// TwinCAT 3 PLC project PulsePower_PLC
// ProgramVersion: 3.1.4023.0
// libraries:
//   Tc2_BACnetRev12, * (Beckhoff Automation GmbH)
//   Tc2_DataExchange, * (Beckhoff Automation GmbH)
//   Tc2_Math, * (Beckhoff Automation GmbH)
//   Tc2_NC, * (Beckhoff Automation GmbH)
//   Tc2_Standard, * (Beckhoff Automation GmbH)
//   Tc2_System, * (Beckhoff Automation GmbH)
//   Tc3_EventLogger, * (Beckhoff Automation GmbH)
//   Tc3_Module, * (Beckhoff Automation GmbH)
// project tree:
//   DUTs/ E_Command.TcDUT (not stored), E_PulseState.TcDUT (not stored), E_Status.TcDUT (not stored), ST_Alarm_Base.TcDUT, ST_Charger_Base.TcDUT (not stored), ST_ChargeTime.TcDUT, ST_Control.TcDUT (not stored), ST_Echo_MCP.TcDUT, ST_Echo_Section.TcDUT (not stored), ST_FieldDevices_Base.TcDUT (not stored), ST_FieldDevices_Form.TcDUT, ST_InstrumentReading.TcDUT (not stored), ST_Recipe.TcDUT (not stored), ST_RelayFaults_Base.TcDUT, ST_RelayFaults_Form.TcDUT, ST_Section_Base.TcDUT, ST_Setpoints_Base.TcDUT, ST_Trip_Base.TcDUT, ST_VoltageFeedback.TcDUT
//   GVLs/ Alarms_DB.TcGVL (not stored), ChargeTime_DB.TcGVL, Command.TcGVL, EngVal.TcGVL, GVL.TcGVL, Recipe.TcGVL, Setpoints.TcGVL (not stored), TxMainPLC.TcGVL, HMI_DB.TcGVL, Input.TcGVL (not stored), InstrumentReading.TcGVL (not stored), LCP.TcGVL, MCP_IO.TcGVL (not stored), Output.TcGVL (not stored), Permissives_DB.TcGVL (not stored), Trips_DB.TcGVL (not stored)
//   / PlcTask.TcTTO (not stored)
//   POUs/ ADC_10V.TcPOU (not stored), ADC_5V.TcPOU (not stored), Alarms.TcPOU, Alarms_FB.TcPOU (not stored), Alias.TcPOU (not stored), AnalogConversion.TcPOU, AQ.TcPOU (not stored), ChargeTime.TcPOU, Communication.TcPOU (not stored), Dump_FB.TcPOU, Heartbeat.TcPOU (not stored), HMI.TcPOU, LCA_CAL.TcPOU (not stored), MAIN.TcPOU, Norm_x.TcPOU (not stored), Permissives.TcPOU, PWMO.TcPOU (not stored), Sequence.TcPOU, Trips.TcPOU
// real-time tasks:
//   TASK PlcTask: cycle T#10ms, priority 20, ADS port 350
// I/O:
//   DEVICE Device 3 (EtherCAT) (disabled), AmsNetId 5.104.224.86.4.1
//   DEVICE Device 1 (EL6751) (disabled), AmsNetId 5.104.224.86.2.1
//   DEVICE Device 2 (EtherCAT), AmsNetId 5.104.224.86.3.1
//     Term 1 (EK1200) [EK1200-5000 EtherCAT Power supply (2A E-Bus)]
//       Term 9 (EL2008) [EL2008 8Ch. Dig. Output 24V, 0.5A]
//       Term 3 (EL9011) [EL9011 End Terminal]
// variable links:
//   PulsePower_PLC/PulsePower_PLC Instance <-> Device 2 (EtherCAT)/Term 1 (EK1200)/Term 9 (EL2008)
//     PlcTask Outputs/Output.R2_01_00 <-> Channel 1/Output

// ---- DUTs/ST_Alarm_Base.TcDUT
TYPE ST_Alarm_Base :
STRUCT
	AlarmWord : WORD;
END_STRUCT
END_TYPE

// ---- DUTs/ST_ChargeTime.TcDUT
TYPE ST_ChargeTime :
STRUCT
	timeToChargeLoad : REAL;
	Power			 : REAL;
END_STRUCT
END_TYPE

// ---- DUTs/ST_Echo_MCP.TcDUT
TYPE ST_Echo_MCP :
STRUCT
	VoltageFeedback : REAL; //DINT;
	CurrentFeedback : REAL; //DINT;
	TDKLoad			: ST_ChargeTime;
	
END_STRUCT
END_TYPE

// ---- DUTs/ST_FieldDevices_Form.TcDUT
TYPE ST_FieldDevices_Form EXTENDS ST_FieldDevices_Base :
STRUCT
	PreFormChargeRly_close		: BOOL;
	FormTrigChargeRly_close		: BOOL;
	PreFormTrigChargeRly_close 	: BOOL;
	PreFormDumpRly_close		: BOOL;
	FormTrigDumpRly1_close		: BOOL;
	PreFormTrigDumpRly1_close	: BOOL;
	
	ClosePreFormChargeRly		: BOOL;
	CloseFormTrigChargeRly		: BOOL;
	ClosePreFormTrigChargeRly	: BOOL;
	OpenPreFormDumpRly			: BOOL;
	OpenFormTrigDumpRly1		: BOOL;
	OpenPreFormTrigDumpRly1		: BOOL;
	
	FormTrigShortContact_close		: BOOL;
	FormTrigUnshortContact_close	: BOOL;
	FormTrigShortContactEngaged		: BOOL;
	FormTrigShortContactUnknown		: BOOL;
	
	PreFormTrigShortContact_close 	: BOOL;
	PreFormTrigUnShortContact_close : BOOL;
	PreFormTrigShortContactEngaged	: BOOL;
	PreFormTrigShortContactUnknown	: BOOL;
	

END_STRUCT
END_TYPE

// ---- DUTs/ST_RelayFaults_Base.TcDUT
TYPE ST_RelayFaults_Base :
STRUCT
	DumpRelay1_FailtoClose		: BOOL;
	DumpRelay1_FailtoOpen		: BOOL;
	DumpRelay1_Failed			: BOOL;
	DumpRly1FaultDelay_TON 		: TON;
	DumpRly2FaultDelay_TON 		: TON;
	
	DumpRelay2_FailtoClose		: BOOL;
	DumpRelay2_FailtoOpen		: BOOL;
	DumpRelay2_Failed			: BOOL;
	
	ChargeRelay1_FailtoClose	: BOOL;
	ChargeRelay1_FailtoOpen		: BOOL;
	ChargeRelay1_Failed			: BOOL;
	ChrgRly1FaultDelay_TON	 	: TON;
	
	ChargeRelay2_FailtoClose	: BOOL;
	ChargeRelay2_FailtoOpen		: BOOL;
	ChargeRelay2_Failed			: BOOL;
	ChrgRly2FaultDelay_TON	 	: TON;
	

END_STRUCT
END_TYPE

// ---- DUTs/ST_RelayFaults_Form.TcDUT
TYPE ST_RelayFaults_Form EXTENDS ST_RelayFaults_Base :
STRUCT
	PreFormChrgRlyFailed				: BOOL;
	PreFormChrgRlyFaultDelay_TON		: TON;
	FormTrigChrgRlyFailed				: BOOL;
	FormTrigChrgRlyFaultDelay_TON		: TON;
	PreFormTrigChrgRlyFailed			: BOOL;
	PreFormTrigChrgRlyFaultDelay_TON	: TON;
	PreFormDumpRlyFailed				: BOOL;
	PreFormDumpRlyFaultDelay_TON		: TON;
	FormTrigDumpRly1Failed				: BOOL;
	FormTrigDumpRlyFaultDelay_TON		: TON;
	PreFormTrigDumpRly1Failed			: BOOL;
	PreFormTrigDumpRlyFaultDelay_TON	: TON;
	
END_STRUCT
END_TYPE

// ---- DUTs/ST_Section_Base.TcDUT
//Base coil type with all the Common functionality
TYPE ST_Section_Base :
STRUCT
	
	Peak : ST_FieldDevices_Base;
	Sust : ST_FieldDevices_Base;
	Form : ST_FieldDevices_Form;
	
	PreFormCapVoltage_raw			: INT;
	PreFormCapVoltage_norm			: REAL;
	PreFormCapVoltageFeedback		: REAL;
	
	FormTriggerVoltage_raw			: INT;
	FormTriggerVoltage_norm			: REAL;
	FormTriggerVoltageFeedback		: REAL;
	
	PreFormTriggerVoltage_raw		: INT;
	PreFormTriggerVoltage_norm		: REAL;
	PreFormTriggerVoltageFeedback	: REAL;
	
	PreFormCapDischarged			: BOOL;
	PreFormCapFullyChaged			: BOOL;
	
	PSU1_DCOK						: BOOL := FALSE;
	//Local_EstopPB_Pressed			: BOOL;  //NC
	SystemReadyToCharge				: BOOL := FALSE;
	LossPneumaticPressure			: BOOL;
	AllCapsDischarged				: BOOL;
	AllCapsFullyCharged				: BOOL;
	//PreFormBank						: ST_ChargeTime;
END_STRUCT
END_TYPE

// ---- DUTs/ST_Setpoints_Base.TcDUT
TYPE ST_Setpoints_Base :
STRUCT
	RequiredChargedV : REAL := 12;
	TotalCapacitance : REAL := 10; //uF - LOCAL ONLY, NOT FROM MAIN PLC - LoadCapacitance
	PSratedV		 : REAL := 50;
	wLCA			 : BOOL := TRUE;
	NumOfCharger	 : INT := 1;
END_STRUCT
END_TYPE

// ---- DUTs/ST_Trip_Base.TcDUT
TYPE ST_Trip_Base :
STRUCT
	ChargerVoltageReadingFaulted 		: BOOL;
	CurrentReadingFaulted 		 		: BOOL;
	
	//ACInterlockRelayFailedtoClose		: BOOL;
	//ACInterlockRelayFailedtoOpen 		: BOOL;
	//ACintLockRlyCloseFaultDelay_TON	: TON;
	//ACintLockRlyOpenFaultDelay_TON	: TON;
	
	Peak 								: ST_RelayFaults_Base;
	Sust 								: ST_RelayFaults_Base;
	Form 								: ST_RelayFaults_Form;
	
	SystemTripped						: BOOL;
	LossPneumaticPressure				: BOOL;
	LossDCPower							: BOOL;
	
	(*HVisoRelayFailedToOpen		: BOOL;
	HVRelayOpenFaultDelay_TON	: TON;
	HVisoRelayFailedToClose		: BOOL;
	HVRelayCloseFaultDelay_TON	: TON;
	*)
END_STRUCT
END_TYPE

// ---- DUTs/ST_VoltageFeedback.TcDUT
TYPE ST_VoltageFeedback :
STRUCT
	voltageFeedback_raw : INT;
END_STRUCT
END_TYPE

// ---- GVLs/ChargeTime_DB.TcGVL
{attribute 'qualified_only'}
VAR_GLOBAL RETAIN
	ChargerDelay_TON : ARRAY[1..8] OF TON;
	ChargerDelay_PT  : ARRAY[1..8] OF TIME;
	ChargerDelay_ET  : ARRAY[1..8] OF TIME;	
	
	//SustChargeTime_TON : ARRAY[1..3] OF TON;
	//SustChargeTime_PT  : ARRAY[1..3] OF TIME;
	//SustChargeTime_ET  : ARRAY[1..3] OF TIME;	
	
	//FormChargeTime_TON : ARRAY[1..2] OF TON;
	//FormChargeTime_PT  : ARRAY[1..2] OF TIME;
	//FormChargeTime_ET  : ARRAY[1..2] OF TIME;
	
	PreFormChargeTime_TON : TON;
	PreFormChargeTime_PT : TIME;
	PreFormChargeTime_ET : TIME;
	
	LongestChargeTime_TON : TON;
	LongestChargeTime_PT : TIME;
	LongestChargeTime_ET : TIME;

	ChargeTimeStartDelay	: ARRAY[1..8] OF INT;
	ChargingTimeElapse		: ARRAY[1..8] OF INT;	
	ChargingTimeElapse_TON	: ARRAY[1..8] OF TON;
	
	PreFormChargeTimeStartDelay : INT;
	PreFormChargingTimeElapse : INT;
	PreFormChargingTimeElapse_TON : TON;
END_VAR

// ---- GVLs/Command.TcGVL
{attribute 'qualified_only'}
VAR_GLOBAL
	eCommand : E_Command;
END_VAR

// ---- GVLs/EngVal.TcGVL
{attribute 'qualified_only'}
VAR_GLOBAL
	Max_50kVChargerVoltage : REAL := 50000; //50kV
	Min_50kVChargerVoltage : REAL := 0;
	
	Max_50kVChargerCurrent : REAL := 0.18; //total peak charge current is 0.18A
	Min_50kVChargerCurrent : REAL := 0;
	
	Max_12kVChargerVoltage : REAL := 12000; //12kV
	Min_12kVChargerVoltage : REAL := 0;
	
	Max_12kVChargerCurrent : REAL := 0.75; //total peak charge current is 0.75A
	Min_12kVChargerCurrent : REAL := 0;
	
	Max_GLS1_ChargerV	   : REAL := 50000; //form trigger
	Max_GLS2_ChargerV	   : REAL := 50000; // preform trigger
	Max_GLS3_ChargerV	   : REAL := 30000; // preform cap charger
	
	Max_CapVoltage			: REAL := 32000;  //assuming 32kV cap....  
	Min_CapVoltage			: REAL := 0;
	
	UpperLimit12kVCaps		: REAL := 10000; //peak and sust
	//LowerLimit12kVCaps	: REAL := -2000;
	UpperLimit50kVCaps		: REAL := 35000; //formation
	
	(*ULimit_PeakCapRequiredV	: REAL := 10000; //10kV veto
	LLimit_PeakCapRequiredV	: REAL := -2000; //-2kV
	ULimit_SustCapRequiredV	: REAL := 12000; //12kv veto
	LLimit_SustCapRequiredV	: REAL := -2000; //-2kv
	ULimit_FormCapRequiredV : REAL := 35000;
	LLimit_FormCapRequiredV : REAL := 0;
	*)
	ULimit_PreFormCapRequiredV : REAL := 30000; //gls3
	LLimit_PreFormCapRequiredV : REAL := 0;
		
END_VAR

// ---- GVLs/GVL.TcGVL
{attribute 'qualified_only'}
VAR_GLOBAL
	alarm_test	: BOOL;
	test		: BOOL;
	RemoteModeSelected : BOOL;
END_VAR

// ---- GVLs/Recipe.TcGVL
{attribute 'qualified_only'}
VAR_GLOBAL
	TDKLoad : ARRAY [1..8] OF ST_Recipe;
	GLSLoad : ST_Recipe;
	GLS1_VSP : REAL := 50; //DINT;
	GLS2_VSP : REAL := 50; //DINT;
	PeakSupplyEN	: BOOL := TRUE;
	SustSupplyEN	: BOOL := TRUE;
	FormSupplyEN	: BOOL := TRUE;
	PFormSupplyEN	: BOOL := TRUE;
END_VAR

// ---- GVLs/TxMainPLC.TcGVL
{attribute 'qualified_only'}
VAR_GLOBAL
	Charger		: ARRAY[1..8] OF ST_Echo_MCP;
	GLSLoad		: ST_ChargeTime;
	Section 	: ARRAY[1..4] OF ST_Echo_Section;
	ChargeRunOutTime	: REAL; //DINT;
	ChargingRunOutTime	: REAL; //DINT;
END_VAR

// ---- GVLs/HMI_DB.TcGVL
{attribute 'qualified_only'}
VAR_GLOBAL PERSISTENT
	RemoteModeSelected 	: BOOL := TRUE;
	
	OpenAllDumpRlyPB	: BOOL;
	CloseAllChargeRlyPB	: BOOL;
	AbortPB				: BOOL;
	
	ChargerHVOFF_rlyDelayPT		: TIME := T#25MS;
	ChargerHVOFF_rlyDelayPT_INT	: INT := 25;
	
	HVONdelayPT					: TIME := T#250MS;
	HVONdelayPT_INT				: INT := 250;
	
	RunOutTMR_PT				: TIME := T#10S;
	RunOutTMR_PT_INT			: INT := 10;
	RunOutTMR_elapse			: INT;
	
	ChargingRunOutTMR_elapse	: INT;
	
	//admin bypasses
	SafetyOKBP					: BOOL;
	AllDumpRelaysOpenBP			: BOOL;
	InterlockPressureLossBP		: BOOL;
	AllChargeRelayCloseBP		: BOOL;
	NoFaultDetectedBP			: BOOL;
	//AllShortingSysRemovedBP		: BOOL;
	AlldcPSUokBP				: BOOL;
	LossHVsignalBP				: BOOL;
	
	//timeToChargeLoad 			: ARRAY [1..8] OF REAL;
	//GLSchargeTime	 			: ARRAY [1..3] OF REAL;
	TDKLoad 					: ARRAY [1..8] OF ST_Setpoints_Base; //or RETAIN
	GLSLoad	 					: ST_Setpoints_Base;
	
	(*PSratedV					: REAL := 50;
	RequiredChargeV				: REAL := 30;
	LoadCapacitance				: REAL := 600;
	wLCA						: BOOL := TRUE;
	NumOfCharger				: INT := 1;*)
END_VAR

VAR_GLOBAL
	LiftMachineGNDsw			: BOOL := FALSE;
	//for startup run
	PeakChargerSP				: DINT;
	SustChargerSP				: DINT;
	FormChargerSP				: DINT;
	PreFormChargerSP			: DINT;
	FormTrigChargerSP			: DINT;
	PreFormTrigChargerSP		: DINT;
	
	OpenAllPeakDumpRlySW		: BOOL := FALSE;
	OpenAllSustDumpRlySW		: BOOL := FALSE;
	OpenAllFormDumpRlySW		: BOOL := FALSE;
	OpenAllPreFormDumpRlySW		: BOOL := FALSE;
	OpenFormTrigDumpRlySW		: BOOL := FALSE;
	OpenPreFormTrigDumpRlySW	: BOOL := FALSE;
	
	CloseAllPeakChargRlySW		: BOOL := FALSE;
	CloseAllSustChargRlySW		: BOOL := FALSE;
	CloseAllFormChargRlySW		: BOOL := FALSE;
	CloseAllPreFormChargRlySW	: BOOL := FALSE;
	CloseFormTrigChargeRlySW	: BOOL := FALSE;
	ClosePreFormTrigChargeRlySW : BOOL := FALSE;
	
	PeakHVONsw					: BOOL := FALSE; //enable
	SustHVONsw					: BOOL := FALSE; //enable
	FormHVONsw					: BOOL := FALSE; //enable
	PreFormHVONsw				: BOOL := FALSE;
	GLS1HVONsw					: BOOL := FALSE;
	GLS2HVONsw					: BOOL := FALSE;
	
	DumpALLPB_Local				: BOOL := FALSE;
	
	(*PeakInhibitONsw				: BOOL;
	SustInhibitONsw				: BOOL;
	FormInhibitONsw				: BOOL;
	PreFormInhibitONsw			: BOOL;
	*)	
END_VAR

// ---- GVLs/LCP.TcGVL
{attribute 'qualified_only'}
VAR_GLOBAL
	Section : ARRAY [1..4] OF ST_Section_Base;
END_VAR

// ---- POUs/Alarms.TcPOU
PROGRAM Alarms
VAR
	bWarning : BOOL;
	bConfirm : BOOL;
	alarms : ARRAY[0..128] OF Alarms_FB;
	
END_VAR

// Alarm Word 1 - MCP Alarms
//MCP Alarms

Alarms_DB.MCP.AlarmWord.0 := Trips_DB.MasterStopPBPressed;
Alarms_DB.MCP.AlarmWord.1 := Trips_DB.CageEStopCircuitBroken;
Alarms_DB.MCP.AlarmWord.2 := Trips_DB.LocalModeSelected;
Alarms_DB.MCP.AlarmWord.3 := Trips_DB.MCPLossDCpower;
Alarms_DB.MCP.AlarmWord.4 := MCP_IO.Charger[1].SummaryFaulted;
Alarms_DB.MCP.AlarmWord.5 := MCP_IO.Charger[2].SummaryFaulted;
Alarms_DB.MCP.AlarmWord.6 := MCP_IO.Charger[3].SummaryFaulted;
Alarms_DB.MCP.AlarmWord.7 := MCP_IO.Charger[4].SummaryFaulted;
Alarms_DB.MCP.AlarmWord.8 := MCP_IO.Charger[5].SummaryFaulted;
Alarms_DB.MCP.AlarmWord.9 := MCP_IO.Charger[6].SummaryFaulted;
Alarms_DB.MCP.AlarmWord.10 := MCP_IO.Charger[7].SummaryFaulted;
Alarms_DB.MCP.AlarmWord.11 := MCP_IO.Charger[8].SummaryFaulted;
Alarms_DB.MCP.AlarmWord.12 := Trips_DB.ChargedTimerRunout;
Alarms_DB.MCP.AlarmWord.13 := Trips_DB.ChargingTimerRunout;
Alarms_DB.MCP.AlarmWord.14 := Trips_DB.MCPsystemTripped;
Alarms_DB.MCP.AlarmWord.15 := Trips_DB.AnyEstopPressed;

//Alarm Word 1 msg
//IE: alarms[299](evtEntry:= Tc_Events.AlarmWord11.b4, bEvt:= gvl.test, bConfirm:= bConfirm);
alarms[0](evtEntry:= Tc_Events.AlarmWord1.b0, bEvt:= Alarms_DB.MCP.AlarmWord.0, bConfirm:= bConfirm);
alarms[1](evtEntry:= Tc_Events.AlarmWord1.b1, bEvt:= Alarms_DB.MCP.AlarmWord.1, bConfirm:= bConfirm);
alarms[2](evtEntry:= Tc_Events.AlarmWord1.b2, bEvt:= Alarms_DB.MCP.AlarmWord.2, bConfirm:= bConfirm);
alarms[3](evtEntry:= Tc_Events.AlarmWord1.b3, bEvt:= Alarms_DB.MCP.AlarmWord.3, bConfirm:= bConfirm);
alarms[4](evtEntry:= Tc_Events.AlarmWord1.b4, bEvt:= Alarms_DB.MCP.AlarmWord.4, bConfirm:= bConfirm);
alarms[5](evtEntry:= Tc_Events.AlarmWord1.b5, bEvt:= Alarms_DB.MCP.AlarmWord.5, bConfirm:= bConfirm);
alarms[6](evtEntry:= Tc_Events.AlarmWord1.b6, bEvt:= Alarms_DB.MCP.AlarmWord.6, bConfirm:= bConfirm);
alarms[7](evtEntry:= Tc_Events.AlarmWord1.b7, bEvt:= Alarms_DB.MCP.AlarmWord.7, bConfirm:= bConfirm);
alarms[8](evtEntry:= Tc_Events.AlarmWord1.b8, bEvt:= Alarms_DB.MCP.AlarmWord.8, bConfirm:= bConfirm);
alarms[9](evtEntry:= Tc_Events.AlarmWord1.b9, bEvt:= Alarms_DB.MCP.AlarmWord.9, bConfirm:= bConfirm);
alarms[0](evtEntry:= Tc_Events.AlarmWord1.b10, bEvt:= Alarms_DB.MCP.AlarmWord.10, bConfirm:= bConfirm);
alarms[11](evtEntry:= Tc_Events.AlarmWord1.b11, bEvt:= Alarms_DB.MCP.AlarmWord.11, bConfirm:= bConfirm);
alarms[12](evtEntry:= Tc_Events.AlarmWord1.b12, bEvt:= Alarms_DB.MCP.AlarmWord.12, bConfirm:= bConfirm);
alarms[13](evtEntry:= Tc_Events.AlarmWord1.b13, bEvt:= Alarms_DB.MCP.AlarmWord.13, bConfirm:= bConfirm);
alarms[14](evtEntry:= Tc_Events.AlarmWord1.b14, bEvt:= Alarms_DB.MCP.AlarmWord.14, bConfirm:= bConfirm);
alarms[15](evtEntry:= Tc_Events.AlarmWord1.b15, bEvt:= Alarms_DB.MCP.AlarmWord.15, bConfirm:= bConfirm);

// Alarm Word 2 - Section 1 Alarms
Alarms_DB.Section1.AlarmWord.0 := Trips_DB.Section[1].SystemTripped;
Alarms_DB.Section1.AlarmWord.1 := Trips_DB.Section[1].LossPneumaticPressure;
Alarms_DB.Section1.AlarmWord.2 := Trips_DB.Section[1].Peak.ChargeRelay1_Failed;
Alarms_DB.Section1.AlarmWord.3 := Trips_DB.Section[1].Peak.ChargeRelay2_Failed;
Alarms_DB.Section1.AlarmWord.4 := Trips_DB.Section[1].Peak.DumpRelay1_Failed;
Alarms_DB.Section1.AlarmWord.5 := Trips_DB.Section[1].Peak.DumpRelay2_Failed;
Alarms_DB.Section1.AlarmWord.6 := Trips_DB.Section[1].Sust.ChargeRelay1_Failed;
Alarms_DB.Section1.AlarmWord.7 := Trips_DB.Section[1].Sust.ChargeRelay2_Failed;
Alarms_DB.Section1.AlarmWord.8 := Trips_DB.Section[1].Sust.DumpRelay1_Failed;
Alarms_DB.Section1.AlarmWord.9 := Trips_DB.Section[1].Sust.DumpRelay2_Failed;
Alarms_DB.Section1.AlarmWord.10 := Trips_DB.Section[1].LossDCPower;


// Alarm Word 2 - Msg
alarms[16](evtEntry:= Tc_Events.AlarmWord2.b0, bEvt:= Alarms_DB.Section1.AlarmWord.0, bConfirm:= bConfirm);
alarms[17](evtEntry:= Tc_Events.AlarmWord2.b1, bEvt:= Alarms_DB.Section1.AlarmWord.1, bConfirm:= bConfirm);
alarms[18](evtEntry:= Tc_Events.AlarmWord2.b2, bEvt:= Alarms_DB.Section1.AlarmWord.2, bConfirm:= bConfirm);
alarms[19](evtEntry:= Tc_Events.AlarmWord2.b3, bEvt:= Alarms_DB.Section1.AlarmWord.3, bConfirm:= bConfirm);
alarms[20](evtEntry:= Tc_Events.AlarmWord2.b4, bEvt:= Alarms_DB.Section1.AlarmWord.4, bConfirm:= bConfirm);
alarms[21](evtEntry:= Tc_Events.AlarmWord2.b5, bEvt:= Alarms_DB.Section1.AlarmWord.5, bConfirm:= bConfirm);
alarms[22](evtEntry:= Tc_Events.AlarmWord2.b6, bEvt:= Alarms_DB.Section1.AlarmWord.6, bConfirm:= bConfirm);
alarms[23](evtEntry:= Tc_Events.AlarmWord2.b7, bEvt:= Alarms_DB.Section1.AlarmWord.7, bConfirm:= bConfirm);
alarms[24](evtEntry:= Tc_Events.AlarmWord2.b8, bEvt:= Alarms_DB.Section1.AlarmWord.8, bConfirm:= bConfirm);
alarms[25](evtEntry:= Tc_Events.AlarmWord2.b9, bEvt:= Alarms_DB.Section1.AlarmWord.9, bConfirm:= bConfirm);
alarms[26](evtEntry:= Tc_Events.AlarmWord2.b10, bEvt:= Alarms_DB.Section1.AlarmWord.10, bConfirm:= bConfirm);
//alarms[27] - spare
//alarms[28] - spare
//alarms[29] - spare
//alarms[30] - spare
//alarms[31] - spare


// Alarm Word 3 - Section 2 Alarms
Alarms_DB.Section2.AlarmWord.0 := Trips_DB.Section[2].SystemTripped;
Alarms_DB.Section2.AlarmWord.1 := Trips_DB.Section[2].LossPneumaticPressure;
Alarms_DB.Section2.AlarmWord.2 := Trips_DB.Section[2].Peak.ChargeRelay1_Failed;
Alarms_DB.Section2.AlarmWord.3 := Trips_DB.Section[2].Peak.ChargeRelay2_Failed;
Alarms_DB.Section2.AlarmWord.4 := Trips_DB.Section[2].Peak.DumpRelay1_Failed;
Alarms_DB.Section2.AlarmWord.5 := Trips_DB.Section[2].Peak.DumpRelay2_Failed;
Alarms_DB.Section2.AlarmWord.6 := Trips_DB.Section[2].Sust.ChargeRelay1_Failed;
Alarms_DB.Section2.AlarmWord.7 := Trips_DB.Section[2].Sust.ChargeRelay2_Failed;
Alarms_DB.Section2.AlarmWord.8 := Trips_DB.Section[2].Sust.DumpRelay1_Failed;
Alarms_DB.Section2.AlarmWord.9 := Trips_DB.Section[2].Sust.DumpRelay2_Failed;
Alarms_DB.Section2.AlarmWord.10 := Trips_DB.Section[2].LossDCPower;


// Alarm Word 3 - Msg
alarms[32](evtEntry:= Tc_Events.AlarmWord3.b0, bEvt:= Alarms_DB.Section2.AlarmWord.0, bConfirm:= bConfirm);
alarms[33](evtEntry:= Tc_Events.AlarmWord3.b1, bEvt:= Alarms_DB.Section2.AlarmWord.1, bConfirm:= bConfirm);
alarms[34](evtEntry:= Tc_Events.AlarmWord3.b2, bEvt:= Alarms_DB.Section2.AlarmWord.2, bConfirm:= bConfirm);
alarms[35](evtEntry:= Tc_Events.AlarmWord3.b3, bEvt:= Alarms_DB.Section2.AlarmWord.3, bConfirm:= bConfirm);
alarms[36](evtEntry:= Tc_Events.AlarmWord3.b4, bEvt:= Alarms_DB.Section2.AlarmWord.4, bConfirm:= bConfirm);
alarms[37](evtEntry:= Tc_Events.AlarmWord3.b5, bEvt:= Alarms_DB.Section2.AlarmWord.5, bConfirm:= bConfirm);
alarms[38](evtEntry:= Tc_Events.AlarmWord3.b6, bEvt:= Alarms_DB.Section2.AlarmWord.6, bConfirm:= bConfirm);
alarms[39](evtEntry:= Tc_Events.AlarmWord3.b7, bEvt:= Alarms_DB.Section2.AlarmWord.7, bConfirm:= bConfirm);
alarms[40](evtEntry:= Tc_Events.AlarmWord3.b8, bEvt:= Alarms_DB.Section2.AlarmWord.8, bConfirm:= bConfirm);
alarms[41](evtEntry:= Tc_Events.AlarmWord3.b9, bEvt:= Alarms_DB.Section2.AlarmWord.9, bConfirm:= bConfirm);
alarms[42](evtEntry:= Tc_Events.AlarmWord3.b10, bEvt:= Alarms_DB.Section2.AlarmWord.10, bConfirm:= bConfirm);
//alarms[43] - spare
//alarms[44] - spare
//alarms[45] - spare
//alarms[46] - spare
//alarms[47] - spare

// Alarm Word 4 - Section 3 Alarms
Alarms_DB.Section3.AlarmWord.0 := Trips_DB.Section[3].SystemTripped;
Alarms_DB.Section3.AlarmWord.1 := Trips_DB.Section[3].LossPneumaticPressure;
Alarms_DB.Section3.AlarmWord.2 := Trips_DB.Section[3].Peak.ChargeRelay1_Failed;
Alarms_DB.Section3.AlarmWord.3 := Trips_DB.Section[3].Peak.ChargeRelay2_Failed;
Alarms_DB.Section3.AlarmWord.4 := Trips_DB.Section[3].Peak.DumpRelay1_Failed;
Alarms_DB.Section3.AlarmWord.5 := Trips_DB.Section[3].Peak.DumpRelay2_Failed;
Alarms_DB.Section3.AlarmWord.6 := Trips_DB.Section[3].Sust.ChargeRelay1_Failed;
Alarms_DB.Section3.AlarmWord.7 := Trips_DB.Section[3].Sust.ChargeRelay2_Failed;
Alarms_DB.Section3.AlarmWord.8 := Trips_DB.Section[3].Sust.DumpRelay1_Failed;
Alarms_DB.Section3.AlarmWord.9 := Trips_DB.Section[3].Sust.DumpRelay2_Failed;
Alarms_DB.Section3.AlarmWord.10 := Trips_DB.Section[3].LossDCPower;


// Alarm Word 4 - Msg
alarms[48](evtEntry:= Tc_Events.AlarmWord4.b0, bEvt:= Alarms_DB.Section3.AlarmWord.0, bConfirm:= bConfirm);
alarms[49](evtEntry:= Tc_Events.AlarmWord4.b1, bEvt:= Alarms_DB.Section3.AlarmWord.1, bConfirm:= bConfirm);
alarms[50](evtEntry:= Tc_Events.AlarmWord4.b2, bEvt:= Alarms_DB.Section3.AlarmWord.2, bConfirm:= bConfirm);
alarms[51](evtEntry:= Tc_Events.AlarmWord4.b3, bEvt:= Alarms_DB.Section3.AlarmWord.3, bConfirm:= bConfirm);
alarms[52](evtEntry:= Tc_Events.AlarmWord4.b4, bEvt:= Alarms_DB.Section3.AlarmWord.4, bConfirm:= bConfirm);
alarms[53](evtEntry:= Tc_Events.AlarmWord4.b5, bEvt:= Alarms_DB.Section3.AlarmWord.5, bConfirm:= bConfirm);
alarms[54](evtEntry:= Tc_Events.AlarmWord4.b6, bEvt:= Alarms_DB.Section3.AlarmWord.6, bConfirm:= bConfirm);
alarms[55](evtEntry:= Tc_Events.AlarmWord4.b7, bEvt:= Alarms_DB.Section3.AlarmWord.7, bConfirm:= bConfirm);
alarms[56](evtEntry:= Tc_Events.AlarmWord4.b8, bEvt:= Alarms_DB.Section3.AlarmWord.8, bConfirm:= bConfirm);
alarms[57](evtEntry:= Tc_Events.AlarmWord4.b9, bEvt:= Alarms_DB.Section3.AlarmWord.9, bConfirm:= bConfirm);
alarms[58](evtEntry:= Tc_Events.AlarmWord4.b10, bEvt:= Alarms_DB.Section3.AlarmWord.10, bConfirm:= bConfirm);
//alarms[59] - spare
//alarms[60] - spare
//alarms[61] - spare
//alarms[62] - spare
//alarms[63] - spare

// Alarm Word 5 - Section 4 Alarms
Alarms_DB.Section4.AlarmWord.0 := Trips_DB.Section[4].SystemTripped;
Alarms_DB.Section4.AlarmWord.1 := Trips_DB.Section[4].LossPneumaticPressure;
Alarms_DB.Section4.AlarmWord.2 := Trips_DB.Section[4].Form.ChargeRelay1_Failed;
Alarms_DB.Section4.AlarmWord.3 := Trips_DB.Section[4].Form.ChargeRelay2_Failed;
Alarms_DB.Section4.AlarmWord.4 := Trips_DB.Section[4].Form.DumpRelay1_Failed;
Alarms_DB.Section4.AlarmWord.5 := Trips_DB.Section[4].Form.DumpRelay2_Failed;
Alarms_DB.Section4.AlarmWord.6 := Trips_DB.Section[4].Form.PreFormChrgRlyFailed;
Alarms_DB.Section4.AlarmWord.7 := Trips_DB.Section[4].Form.FormTrigChrgRlyFailed;
Alarms_DB.Section4.AlarmWord.8 := Trips_DB.Section[4].Form.PreFormTrigChrgRlyFailed;
Alarms_DB.Section4.AlarmWord.9 := Trips_DB.Section[4].Form.PreFormDumpRlyFailed;
Alarms_DB.Section4.AlarmWord.10 := Trips_DB.Section[4].Form.FormTrigDumpRly1Failed;
Alarms_DB.Section4.AlarmWord.11 := Trips_DB.Section[4].Form.PreFormTrigDumpRly1Failed;
Alarms_DB.Section4.AlarmWord.12 := Trips_DB.Section[4].LossDCPower;

// Alarm Word 5 - Msg
alarms[64](evtEntry:= Tc_Events.AlarmWord5.b0, bEvt:= Alarms_DB.Section4.AlarmWord.0, bConfirm:= bConfirm);
alarms[65](evtEntry:= Tc_Events.AlarmWord5.b1, bEvt:= Alarms_DB.Section4.AlarmWord.1, bConfirm:= bConfirm);
alarms[66](evtEntry:= Tc_Events.AlarmWord5.b2, bEvt:= Alarms_DB.Section4.AlarmWord.2, bConfirm:= bConfirm);
alarms[67](evtEntry:= Tc_Events.AlarmWord5.b3, bEvt:= Alarms_DB.Section4.AlarmWord.3, bConfirm:= bConfirm);
alarms[68](evtEntry:= Tc_Events.AlarmWord5.b4, bEvt:= Alarms_DB.Section4.AlarmWord.4, bConfirm:= bConfirm);
alarms[69](evtEntry:= Tc_Events.AlarmWord5.b5, bEvt:= Alarms_DB.Section4.AlarmWord.5, bConfirm:= bConfirm);
alarms[70](evtEntry:= Tc_Events.AlarmWord5.b6, bEvt:= Alarms_DB.Section4.AlarmWord.6, bConfirm:= bConfirm);
alarms[71](evtEntry:= Tc_Events.AlarmWord5.b7, bEvt:= Alarms_DB.Section4.AlarmWord.7, bConfirm:= bConfirm);
alarms[72](evtEntry:= Tc_Events.AlarmWord5.b8, bEvt:= Alarms_DB.Section4.AlarmWord.8, bConfirm:= bConfirm);
alarms[73](evtEntry:= Tc_Events.AlarmWord5.b9, bEvt:= Alarms_DB.Section4.AlarmWord.9, bConfirm:= bConfirm);
alarms[74](evtEntry:= Tc_Events.AlarmWord5.b10, bEvt:= Alarms_DB.Section4.AlarmWord.10, bConfirm:= bConfirm);
alarms[75](evtEntry:= Tc_Events.AlarmWord5.b10, bEvt:= Alarms_DB.Section4.AlarmWord.11, bConfirm:= bConfirm);
alarms[76](evtEntry:= Tc_Events.AlarmWord5.b10, bEvt:= Alarms_DB.Section4.AlarmWord.12, bConfirm:= bConfirm);
//alarms[77] - spare
//alarms[78] - spare
//alarms[79] - spare

// Alarm Word 6 - Alarms
Alarms_DB.AlarmWord6.AlarmWord.0:= Trips_DB.Charger[1].OverTemp;
Alarms_DB.AlarmWord6.AlarmWord.1 := Trips_DB.Charger[1].InterlockOpen;
Alarms_DB.AlarmWord6.AlarmWord.2 := Trips_DB.Charger[1].LoadFaulted;
Alarms_DB.AlarmWord6.AlarmWord.3 := Trips_DB.Charger[2].OverTemp;
Alarms_DB.AlarmWord6.AlarmWord.4 := Trips_DB.Charger[2].InterlockOpen;
Alarms_DB.AlarmWord6.AlarmWord.5 := Trips_DB.Charger[2].LoadFaulted;
Alarms_DB.AlarmWord6.AlarmWord.6 := Trips_DB.Charger[3].OverTemp;
Alarms_DB.AlarmWord6.AlarmWord.7 := Trips_DB.Charger[3].InterlockOpen;
Alarms_DB.AlarmWord6.AlarmWord.8 := Trips_DB.Charger[3].LoadFaulted;
Alarms_DB.AlarmWord6.AlarmWord.9 := Trips_DB.Charger[4].OverTemp;
Alarms_DB.AlarmWord6.AlarmWord.10 := Trips_DB.Charger[4].InterlockOpen;
Alarms_DB.AlarmWord6.AlarmWord.11 := Trips_DB.Charger[4].LoadFaulted;
Alarms_DB.AlarmWord6.AlarmWord.12 := Trips_DB.Charger[5].OverTemp;
Alarms_DB.AlarmWord6.AlarmWord.13 := Trips_DB.Charger[5].InterlockOpen;
Alarms_DB.AlarmWord6.AlarmWord.14 := Trips_DB.Charger[5].LoadFaulted;

// Alarm Word 6 - Msg
alarms[80](evtEntry:= Tc_Events.AlarmWord6.b0, bEvt:= Alarms_DB.AlarmWord6.AlarmWord.0, bConfirm:= bConfirm);
alarms[81](evtEntry:= Tc_Events.AlarmWord6.b1, bEvt:= Alarms_DB.AlarmWord6.AlarmWord.1, bConfirm:= bConfirm);
alarms[82](evtEntry:= Tc_Events.AlarmWord6.b2, bEvt:= Alarms_DB.AlarmWord6.AlarmWord.2, bConfirm:= bConfirm);
alarms[83](evtEntry:= Tc_Events.AlarmWord6.b3, bEvt:= Alarms_DB.AlarmWord6.AlarmWord.3, bConfirm:= bConfirm);
alarms[84](evtEntry:= Tc_Events.AlarmWord6.b4, bEvt:= Alarms_DB.AlarmWord6.AlarmWord.4, bConfirm:= bConfirm);
alarms[85](evtEntry:= Tc_Events.AlarmWord6.b5, bEvt:= Alarms_DB.AlarmWord6.AlarmWord.5, bConfirm:= bConfirm);
alarms[86](evtEntry:= Tc_Events.AlarmWord6.b6, bEvt:= Alarms_DB.AlarmWord6.AlarmWord.6, bConfirm:= bConfirm);
alarms[87](evtEntry:= Tc_Events.AlarmWord6.b7, bEvt:= Alarms_DB.AlarmWord6.AlarmWord.7, bConfirm:= bConfirm);
alarms[88](evtEntry:= Tc_Events.AlarmWord6.b8, bEvt:= Alarms_DB.AlarmWord6.AlarmWord.8, bConfirm:= bConfirm);
alarms[89](evtEntry:= Tc_Events.AlarmWord6.b9, bEvt:= Alarms_DB.AlarmWord6.AlarmWord.9, bConfirm:= bConfirm);
alarms[90](evtEntry:= Tc_Events.AlarmWord6.b10, bEvt:= Alarms_DB.AlarmWord6.AlarmWord.10, bConfirm:= bConfirm);
alarms[91](evtEntry:= Tc_Events.AlarmWord6.b11, bEvt:= Alarms_DB.AlarmWord6.AlarmWord.11, bConfirm:= bConfirm);
alarms[92](evtEntry:= Tc_Events.AlarmWord6.b12, bEvt:= Alarms_DB.AlarmWord6.AlarmWord.12, bConfirm:= bConfirm);
//alarms[93]
//alarms[94]
//alarms[95]

// Alarm Word 7 - Charger Alarms
Alarms_DB.AlarmWord7.AlarmWord.0 := Trips_DB.Charger[6].OverTemp;
Alarms_DB.AlarmWord7.AlarmWord.1 := Trips_DB.Charger[6].InterlockOpen;
Alarms_DB.AlarmWord7.AlarmWord.2 := Trips_DB.Charger[6].LoadFaulted;
Alarms_DB.AlarmWord7.AlarmWord.3 := Trips_DB.Charger[7].OverTemp;
Alarms_DB.AlarmWord7.AlarmWord.4 := Trips_DB.Charger[7].InterlockOpen;
Alarms_DB.AlarmWord7.AlarmWord.5 := Trips_DB.Charger[7].LoadFaulted;
Alarms_DB.AlarmWord7.AlarmWord.6 := Trips_DB.Charger[8].OverTemp;
Alarms_DB.AlarmWord7.AlarmWord.7 := Trips_DB.Charger[8].InterlockOpen;
Alarms_DB.AlarmWord7.AlarmWord.8 := Trips_DB.Charger[8].LoadFaulted;
Alarms_DB.AlarmWord7.AlarmWord.9 := Trips_DB.AnyChargerOverTemp; 
Alarms_DB.AlarmWord7.AlarmWord.10 := Trips_DB.AnyChargerLoadFault; 
Alarms_DB.AlarmWord7.AlarmWord.11 := Trips_DB.AnySystemTripped; 
Alarms_DB.AlarmWord7.AlarmWord.12 := Trips_DB.MachineGNDrlyFailed; 
Alarms_DB.AlarmWord7.AlarmWord.13 := Trips_DB.AnyChargeRlyFail; 
Alarms_DB.AlarmWord7.AlarmWord.14 := Trips_DB.AnyDumpRlyFail; 
Alarms_DB.AlarmWord7.AlarmWord.15 := Trips_DB.AnyLossInhibitSignal; 

// Alarm Word 7 - Msg
alarms[96](evtEntry:= Tc_Events.AlarmWord7.b0, bEvt:= Alarms_DB.AlarmWord7.AlarmWord.0, bConfirm:= bConfirm);
alarms[97](evtEntry:= Tc_Events.AlarmWord7.b1, bEvt:= Alarms_DB.AlarmWord7.AlarmWord.1, bConfirm:= bConfirm);
alarms[98](evtEntry:= Tc_Events.AlarmWord7.b2, bEvt:= Alarms_DB.AlarmWord7.AlarmWord.2, bConfirm:= bConfirm);
alarms[99](evtEntry:= Tc_Events.AlarmWord7.b3, bEvt:= Alarms_DB.AlarmWord7.AlarmWord.3, bConfirm:= bConfirm);
alarms[100](evtEntry:= Tc_Events.AlarmWord7.b4, bEvt:= Alarms_DB.AlarmWord7.AlarmWord.4, bConfirm:= bConfirm);
alarms[101](evtEntry:= Tc_Events.AlarmWord7.b5, bEvt:= Alarms_DB.AlarmWord7.AlarmWord.5, bConfirm:= bConfirm);
alarms[102](evtEntry:= Tc_Events.AlarmWord7.b6, bEvt:= Alarms_DB.AlarmWord7.AlarmWord.6, bConfirm:= bConfirm);
alarms[103](evtEntry:= Tc_Events.AlarmWord7.b7, bEvt:= Alarms_DB.AlarmWord7.AlarmWord.7, bConfirm:= bConfirm);
alarms[104](evtEntry:= Tc_Events.AlarmWord7.b8, bEvt:= Alarms_DB.AlarmWord7.AlarmWord.8, bConfirm:= bConfirm);
alarms[105](evtEntry:= Tc_Events.AlarmWord7.b9, bEvt:= Alarms_DB.AlarmWord7.AlarmWord.9, bConfirm:= bConfirm);
alarms[106](evtEntry:= Tc_Events.AlarmWord7.b10, bEvt:= Alarms_DB.AlarmWord7.AlarmWord.10, bConfirm:= bConfirm);
alarms[107](evtEntry:= Tc_Events.AlarmWord7.b11, bEvt:= Alarms_DB.AlarmWord7.AlarmWord.11, bConfirm:= bConfirm);
alarms[108](evtEntry:= Tc_Events.AlarmWord7.b12, bEvt:= Alarms_DB.AlarmWord7.AlarmWord.12, bConfirm:= bConfirm);
alarms[109](evtEntry:= Tc_Events.AlarmWord7.b13, bEvt:= Alarms_DB.AlarmWord7.AlarmWord.13, bConfirm:= bConfirm);
alarms[110](evtEntry:= Tc_Events.AlarmWord7.b14, bEvt:= Alarms_DB.AlarmWord7.AlarmWord.14, bConfirm:= bConfirm);
alarms[111] (evtEntry:= Tc_Events.AlarmWord7.b15, bEvt:= Alarms_DB.AlarmWord7.AlarmWord.15, bConfirm:= bConfirm);


//Alarm Word 8 
Alarms_DB.AlarmWord8.AlarmWord.0 := NOT Trips_DB.AllDCpsuOK;
Alarms_DB.AlarmWord8.AlarmWord.1 := Trips_DB.AnyChargerFaulted;
Alarms_DB.AlarmWord8.AlarmWord.2 := Trips_DB.AnyLossHVONsignal;
Alarms_DB.AlarmWord8.AlarmWord.3 := NOT Trips_DB.NoFaultDetected;
Alarms_DB.AlarmWord8.AlarmWord.4 := LCP.Section[1].Peak.ShortContact1unknown;
Alarms_DB.AlarmWord8.AlarmWord.5 := LCP.Section[1].Peak.ShortContact2unknown;
Alarms_DB.AlarmWord8.AlarmWord.6 := LCP.Section[2].Peak.ShortContact1unknown;
Alarms_DB.AlarmWord8.AlarmWord.7 := LCP.Section[2].Peak.ShortContact2unknown;
Alarms_DB.AlarmWord8.AlarmWord.8 := LCP.Section[3].Peak.ShortContact1unknown;
Alarms_DB.AlarmWord8.AlarmWord.9 := LCP.Section[3].Peak.ShortContact2unknown;
Alarms_DB.AlarmWord8.AlarmWord.10 := LCP.Section[1].Sust.ShortContact1unknown;
Alarms_DB.AlarmWord8.AlarmWord.11 := LCP.Section[1].Sust.ShortContact2unknown;
Alarms_DB.AlarmWord8.AlarmWord.12 := LCP.Section[2].Sust.ShortContact1unknown;
Alarms_DB.AlarmWord8.AlarmWord.13 := LCP.Section[2].Sust.ShortContact2unknown;
Alarms_DB.AlarmWord8.AlarmWord.14 := LCP.Section[3].Sust.ShortContact1unknown;
Alarms_DB.AlarmWord8.AlarmWord.15 := LCP.Section[3].Sust.ShortContact2unknown;

//Alarm Word 8 - msg
alarms[112](evtEntry:= Tc_Events.AlarmWord8.b0, bEvt:= Alarms_DB.AlarmWord8.AlarmWord.0, bConfirm:= bConfirm);
alarms[113](evtEntry:= Tc_Events.AlarmWord8.b1, bEvt:= Alarms_DB.AlarmWord8.AlarmWord.1, bConfirm:= bConfirm);
alarms[114](evtEntry:= Tc_Events.AlarmWord8.b2, bEvt:= Alarms_DB.AlarmWord8.AlarmWord.2, bConfirm:= bConfirm);
alarms[115](evtEntry:= Tc_Events.AlarmWord8.b3, bEvt:= Alarms_DB.AlarmWord8.AlarmWord.3, bConfirm:= bConfirm);
alarms[116](evtEntry:= Tc_Events.AlarmWord8.b4, bEvt:= Alarms_DB.AlarmWord8.AlarmWord.4, bConfirm:= bConfirm);
alarms[117](evtEntry:= Tc_Events.AlarmWord8.b5, bEvt:= Alarms_DB.AlarmWord8.AlarmWord.5, bConfirm:= bConfirm);
alarms[118](evtEntry:= Tc_Events.AlarmWord8.b6, bEvt:= Alarms_DB.AlarmWord8.AlarmWord.6, bConfirm:= bConfirm);
alarms[119](evtEntry:= Tc_Events.AlarmWord8.b7, bEvt:= Alarms_DB.AlarmWord8.AlarmWord.7, bConfirm:= bConfirm);
alarms[120](evtEntry:= Tc_Events.AlarmWord8.b8, bEvt:= Alarms_DB.AlarmWord8.AlarmWord.8, bConfirm:= bConfirm);
alarms[121](evtEntry:= Tc_Events.AlarmWord8.b9, bEvt:= Alarms_DB.AlarmWord8.AlarmWord.9, bConfirm:= bConfirm);
alarms[122](evtEntry:= Tc_Events.AlarmWord8.b10, bEvt:= Alarms_DB.AlarmWord8.AlarmWord.10, bConfirm:= bConfirm);
alarms[123](evtEntry:= Tc_Events.AlarmWord8.b11, bEvt:= Alarms_DB.AlarmWord8.AlarmWord.11, bConfirm:= bConfirm);
alarms[124](evtEntry:= Tc_Events.AlarmWord8.b12, bEvt:= Alarms_DB.AlarmWord8.AlarmWord.12, bConfirm:= bConfirm);
alarms[125](evtEntry:= Tc_Events.AlarmWord8.b13, bEvt:= Alarms_DB.AlarmWord8.AlarmWord.13, bConfirm:= bConfirm);
alarms[126](evtEntry:= Tc_Events.AlarmWord8.b14, bEvt:= Alarms_DB.AlarmWord8.AlarmWord.14, bConfirm:= bConfirm);
alarms[127] (evtEntry:= Tc_Events.AlarmWord8.b15, bEvt:= Alarms_DB.AlarmWord8.AlarmWord.15, bConfirm:= bConfirm);

//Alarm Word 9 
Alarms_DB.AlarmWord9.AlarmWord.0 := LCP.Section[4].Form.ShortContact1unknown;
Alarms_DB.AlarmWord9.AlarmWord.1 := LCP.Section[4].Form.ShortContact2unknown;
Alarms_DB.AlarmWord9.AlarmWord.2 := LCP.Section[4].Form.FormTrigShortContactUnknown;
Alarms_DB.AlarmWord9.AlarmWord.3 := LCP.Section[4].Form.PreFormTrigShortContactUnknown;
Alarms_DB.AlarmWord9.AlarmWord.4 := NOT Permissives_DB.NoShortingUnknowns;
Alarms_DB.AlarmWord9.AlarmWord.5 := NOT Permissives_DB.NoInterlockPressureLoss;
Alarms_DB.AlarmWord9.AlarmWord.6 := NOT Permissives_DB.SafetyOK;
//Alarms_DB.AlarmWord9.AlarmWord.7 := 
//Alarms_DB.AlarmWord9.AlarmWord.8 := 
//Alarms_DB.AlarmWord9.AlarmWord.9 := 
//Alarms_DB.AlarmWord9.AlarmWord.10 := 
//Alarms_DB.AlarmWord9.AlarmWord.11 := 
//Alarms_DB.AlarmWord9.AlarmWord.12 := 
//Alarms_DB.AlarmWord9.AlarmWord.13 := 
//Alarms_DB.AlarmWord9.AlarmWord.14 := 
Alarms_DB.AlarmWord9.AlarmWord.15 := Trips_DB.DumpTimerRunout;

//Alarm Word 9 - msg
alarms[112](evtEntry:= Tc_Events.AlarmWord9.b0, bEvt:= Alarms_DB.AlarmWord9.AlarmWord.0, bConfirm:= bConfirm);
alarms[113](evtEntry:= Tc_Events.AlarmWord9.b1, bEvt:= Alarms_DB.AlarmWord9.AlarmWord.1, bConfirm:= bConfirm);
alarms[114](evtEntry:= Tc_Events.AlarmWord9.b2, bEvt:= Alarms_DB.AlarmWord9.AlarmWord.2, bConfirm:= bConfirm);
alarms[115](evtEntry:= Tc_Events.AlarmWord9.b3, bEvt:= Alarms_DB.AlarmWord9.AlarmWord.3, bConfirm:= bConfirm);
alarms[116](evtEntry:= Tc_Events.AlarmWord9.b4, bEvt:= Alarms_DB.AlarmWord9.AlarmWord.4, bConfirm:= bConfirm);
alarms[117](evtEntry:= Tc_Events.AlarmWord9.b5, bEvt:= Alarms_DB.AlarmWord9.AlarmWord.5, bConfirm:= bConfirm);
alarms[118](evtEntry:= Tc_Events.AlarmWord9.b6, bEvt:= Alarms_DB.AlarmWord9.AlarmWord.6, bConfirm:= bConfirm);
//alarms[119](evtEntry:= Tc_Events.AlarmWord9.b7, bEvt:= Alarms_DB.AlarmWord9.AlarmWord.7, bConfirm:= bConfirm);
//alarms[120](evtEntry:= Tc_Events.AlarmWord9.b8, bEvt:= Alarms_DB.AlarmWord9.AlarmWord.8, bConfirm:= bConfirm);
//alarms[121](evtEntry:= Tc_Events.AlarmWord9.b9, bEvt:= Alarms_DB.AlarmWord9.AlarmWord.9, bConfirm:= bConfirm);
//alarms[122](evtEntry:= Tc_Events.AlarmWord9.b10, bEvt:= Alarms_DB.AlarmWord9.AlarmWord.10, bConfirm:= bConfirm);
//alarms[123](evtEntry:= Tc_Events.AlarmWord9.b11, bEvt:= Alarms_DB.AlarmWord9.AlarmWord.11, bConfirm:= bConfirm);
//alarms[124](evtEntry:= Tc_Events.AlarmWord9.b12, bEvt:= Alarms_DB.AlarmWord9.AlarmWord.12, bConfirm:= bConfirm);
//alarms[125](evtEntry:= Tc_Events.AlarmWord9.b13, bEvt:= Alarms_DB.AlarmWord9.AlarmWord.13, bConfirm:= bConfirm);
//alarms[126](evtEntry:= Tc_Events.AlarmWord9.b14, bEvt:= Alarms_DB.AlarmWord9.AlarmWord.14, bConfirm:= bConfirm);
alarms[127] (evtEntry:= Tc_Events.AlarmWord9.b15, bEvt:= Alarms_DB.AlarmWord9.AlarmWord.15, bConfirm:= bConfirm);

//Alarm Word 11
(* uncomment this when instrument is ready
Alarms_DB.AlarmWord_11.AlarmWord.0 := Devices.Coil1.AC_Interlock_RlyOpen;
Alarms_DB.AlarmWord_11.AlarmWord.1 := Devices.Coil2.AC_Interlock_RlyOpen;
Alarms_DB.AlarmWord_11.AlarmWord.2 := Devices.Coil3.AC_Interlock_RlyOpen;
Alarms_DB.AlarmWord_11.AlarmWord.3 := Devices.Coil4.AC_Interlock_RlyOpen;
Alarms_DB.AlarmWord_11.AlarmWord.4 := Devices.Coil5.AC_Interlock_RlyOpen;
Alarms_DB.AlarmWord_11.AlarmWord.5 := Devices.Coil6.AC_Interlock_RlyOpen;
Alarms_DB.AlarmWord_11.AlarmWord.6 := Devices.Coil7.AC_Interlock_RlyOpen;
Alarms_DB.AlarmWord_11.AlarmWord.7 := Devices.Coil8.AC_Interlock_RlyOpen;
Alarms_DB.AlarmWord_11.AlarmWord.8 := Devices.Coil9.AC_Interlock_RlyOpen;
Alarms_DB.AlarmWord_11.AlarmWord.9 := Devices.Coil10.AC_Interlock_RlyOpen;
Alarms_DB.AlarmWord_11.AlarmWord.10 := NOT Permissives.AllInterlock_Closed;
*)
//Alarm Word 11 - msg
(*alarms[160](evtEntry:= Tc_Events.AlarmWord11.b0, bEvt:= Alarms_DB.AlarmWord_11.AlarmWord.0, bConfirm:= bConfirm);
alarms[161](evtEntry:= Tc_Events.AlarmWord11.b1, bEvt:= Alarms_DB.AlarmWord_11.AlarmWord.1, bConfirm:= bConfirm);
alarms[162](evtEntry:= Tc_Events.AlarmWord11.b2, bEvt:= Alarms_DB.AlarmWord_11.AlarmWord.2, bConfirm:= bConfirm);
alarms[163](evtEntry:= Tc_Events.AlarmWord11.b3, bEvt:= Alarms_DB.AlarmWord_11.AlarmWord.3, bConfirm:= bConfirm);
alarms[164](evtEntry:= Tc_Events.AlarmWord11.b4, bEvt:= Alarms_DB.AlarmWord_11.AlarmWord.4, bConfirm:= bConfirm);
alarms[165](evtEntry:= Tc_Events.AlarmWord11.b5, bEvt:= Alarms_DB.AlarmWord_11.AlarmWord.5, bConfirm:= bConfirm);
alarms[166](evtEntry:= Tc_Events.AlarmWord11.b6, bEvt:= Alarms_DB.AlarmWord_11.AlarmWord.6, bConfirm:= bConfirm);
alarms[167](evtEntry:= Tc_Events.AlarmWord11.b7, bEvt:= Alarms_DB.AlarmWord_11.AlarmWord.7, bConfirm:= bConfirm);
alarms[168](evtEntry:= Tc_Events.AlarmWord11.b8, bEvt:= Alarms_DB.AlarmWord_11.AlarmWord.8, bConfirm:= bConfirm);
alarms[169](evtEntry:= Tc_Events.AlarmWord11.b9, bEvt:= Alarms_DB.AlarmWord_11.AlarmWord.9, bConfirm:= bConfirm);
alarms[170](evtEntry:= Tc_Events.AlarmWord11.b10, bEvt:= Alarms_DB.AlarmWord_11.AlarmWord.10, bConfirm:= bConfirm);

//Alarm Word 12




//Alarm Word 22
//uncomment this when instrument is ready - commented out for testing only
Alarms_DB.AlarmWord_22.AlarmWord.0 := MCP_IO.MasterStopPB_Pressed; //NC
(*//Alarms_DB1.AlarmWord_22.AlarmWord.1 := Devices.Coil[1].Local_EstopPB_Pressed; //NC
Alarms_DB1.AlarmWord_22.AlarmWord.2 := Devices.Coil2.Local_EstopPB_Pressed; //NC
Alarms_DB1.AlarmWord_22.AlarmWord.3 := Devices.Coil3.Local_EstopPB_Pressed; //NC
Alarms_DB1.AlarmWord_22.AlarmWord.4 := Devices.Coil4.Local_EstopPB_Pressed; //NC
Alarms_DB1.AlarmWord_22.AlarmWord.5 := Devices.Coil5.Local_EstopPB_Pressed; //NC
Alarms_DB1.AlarmWord_22.AlarmWord.6 := Devices.Coil6.Local_EstopPB_Pressed; //NC
Alarms_DB1.AlarmWord_22.AlarmWord.7 := Devices.Coil7.Local_EstopPB_Pressed; //NC
Alarms_DB1.AlarmWord_22.AlarmWord.8 := Devices.Coil8.Local_EstopPB_Pressed; //NC
Alarms_DB1.AlarmWord_22.AlarmWord.9 := Devices.Coil9.Local_EstopPB_Pressed; //NC
Alarms_DB1.AlarmWord_22.AlarmWord.10 := Devices.Coil10.Local_EstopPB_Pressed; //NC
//Alarms_DB1.AlarmWord_22.AlarmWord.11 := NOT Input.R1_01_02; //0 = Manual Mode , 1 = Auto mode
//Alarms_DB1.AlarmWord_22.AlarmWord.12 := NOT Input.R1_01_01; //0 = circuit broken , 1 = circuit ok
//Alarms_DB1.AlarmWord_22.AlarmWord.13 := Spare
//Alarms_DB1.AlarmWord_22.AlarmWord.14 := Spare
//Alarms_DB1.AlarmWord_22.AlarmWord.15 := Spare
*)

//Alarm Word 22 msg
alarms[336](evtEntry:= Tc_Events.AlarmWord22.b0, bEvt:= Alarms_DB.AlarmWord_22.AlarmWord.0, bConfirm:= bConfirm);
alarms[337](evtEntry:= Tc_Events.AlarmWord22.b1, bEvt:= Alarms_DB.AlarmWord_22.AlarmWord.1, bConfirm:= bConfirm);
alarms[338](evtEntry:= Tc_Events.AlarmWord22.b2, bEvt:= Alarms_DB.AlarmWord_22.AlarmWord.2, bConfirm:= bConfirm);
alarms[339](evtEntry:= Tc_Events.AlarmWord22.b3, bEvt:= Alarms_DB.AlarmWord_22.AlarmWord.3, bConfirm:= bConfirm);
alarms[340](evtEntry:= Tc_Events.AlarmWord22.b4, bEvt:= Alarms_DB.AlarmWord_22.AlarmWord.4, bConfirm:= bConfirm);
alarms[341](evtEntry:= Tc_Events.AlarmWord22.b5, bEvt:= Alarms_DB.AlarmWord_22.AlarmWord.5, bConfirm:= bConfirm);
alarms[342](evtEntry:= Tc_Events.AlarmWord22.b6, bEvt:= Alarms_DB.AlarmWord_22.AlarmWord.6, bConfirm:= bConfirm);
alarms[343](evtEntry:= Tc_Events.AlarmWord22.b7, bEvt:= Alarms_DB.AlarmWord_22.AlarmWord.7, bConfirm:= bConfirm);
alarms[344](evtEntry:= Tc_Events.AlarmWord22.b8, bEvt:= Alarms_DB.AlarmWord_22.AlarmWord.8, bConfirm:= bConfirm);
alarms[345](evtEntry:= Tc_Events.AlarmWord22.b9, bEvt:= Alarms_DB.AlarmWord_22.AlarmWord.9, bConfirm:= bConfirm);
alarms[346](evtEntry:= Tc_Events.AlarmWord22.b10, bEvt:= Alarms_DB.AlarmWord_22.AlarmWord.10, bConfirm:= bConfirm);
alarms[347](evtEntry:= Tc_Events.AlarmWord22.b11, bEvt:= Alarms_DB.AlarmWord_22.AlarmWord.11, bConfirm:= bConfirm);
alarms[348](evtEntry:= Tc_Events.AlarmWord22.b12, bEvt:= Alarms_DB.AlarmWord_22.AlarmWord.12, bConfirm:= bConfirm);

//Alarm Word 23
(* uncomment when instrument is ready
Alarms_DB.AlarmWord_23.AlarmWord.0 := Trips_DB.Coil[1].ChargeRelay_FailtoClose; 
Alarms_DB.AlarmWord_23.AlarmWord.1 := Trips_DB.Coil[1].ChargeRelay_FailtoOpen;
Alarms_DB.AlarmWord_23.AlarmWord.2 := Trips_DB.Coil[2].ChargeRelay_FailtoClose;
Alarms_DB.AlarmWord_23.AlarmWord.3 := Trips_DB.Coil[2].ChargeRelay_FailtoOpen;
Alarms_DB.AlarmWord_23.AlarmWord.4 := Trips_DB.Coil[3].ChargeRelay_FailtoClose;
Alarms_DB.AlarmWord_23.AlarmWord.5 := Trips_DB.Coil[3].ChargeRelay_FailtoOpen;
Alarms_DB.AlarmWord_23.AlarmWord.6 := Trips_DB.Coil[4].ChargeRelay_FailtoClose;
Alarms_DB.AlarmWord_23.AlarmWord.7 := Trips_DB.Coil[4].ChargeRelay_FailtoOpen;
Alarms_DB.AlarmWord_23.AlarmWord.8 := Trips_DB.Coil[5].ChargeRelay_FailtoClose;
Alarms_DB.AlarmWord_23.AlarmWord.9 := Trips_DB.Coil[5].ChargeRelay_FailtoOpen;
Alarms_DB.AlarmWord_23.AlarmWord.10 := Trips_DB.Coil[6].ChargeRelay_FailtoClose;
Alarms_DB.AlarmWord_23.AlarmWord.11 := Trips_DB.Coil[6].ChargeRelay_FailtoOpen;
Alarms_DB.AlarmWord_23.AlarmWord.12 := Trips_DB.Coil[7].ChargeRelay_FailtoClose;
Alarms_DB.AlarmWord_23.AlarmWord.13 := Trips_DB.Coil[7].ChargeRelay_FailtoOpen;
Alarms_DB.AlarmWord_23.AlarmWord.14 := Trips_DB.Coil[8].ChargeRelay_FailtoClose;
Alarms_DB.AlarmWord_23.AlarmWord.15 := Trips_DB.Coil[9].ChargeRelay_FailtoOpen;
*)
//Alarm Word 23 msg
alarms[352](evtEntry:= Tc_Events.AlarmWord23.b0, bEvt:= Alarms_DB.AlarmWord_23.AlarmWord.0, bConfirm:= bConfirm);
alarms[353](evtEntry:= Tc_Events.AlarmWord23.b1, bEvt:= Alarms_DB.AlarmWord_23.AlarmWord.1, bConfirm:= bConfirm);
alarms[354](evtEntry:= Tc_Events.AlarmWord23.b2, bEvt:= Alarms_DB.AlarmWord_23.AlarmWord.2, bConfirm:= bConfirm);
alarms[355](evtEntry:= Tc_Events.AlarmWord23.b3, bEvt:= Alarms_DB.AlarmWord_23.AlarmWord.3, bConfirm:= bConfirm);
alarms[356](evtEntry:= Tc_Events.AlarmWord23.b4, bEvt:= Alarms_DB.AlarmWord_23.AlarmWord.4, bConfirm:= bConfirm);
alarms[357](evtEntry:= Tc_Events.AlarmWord23.b5, bEvt:= Alarms_DB.AlarmWord_23.AlarmWord.5, bConfirm:= bConfirm);
alarms[358](evtEntry:= Tc_Events.AlarmWord23.b6, bEvt:= Alarms_DB.AlarmWord_23.AlarmWord.6, bConfirm:= bConfirm);
alarms[359](evtEntry:= Tc_Events.AlarmWord23.b7, bEvt:= Alarms_DB.AlarmWord_23.AlarmWord.7, bConfirm:= bConfirm);
alarms[360](evtEntry:= Tc_Events.AlarmWord23.b8, bEvt:= Alarms_DB.AlarmWord_23.AlarmWord.8, bConfirm:= bConfirm);
alarms[361](evtEntry:= Tc_Events.AlarmWord23.b9, bEvt:= Alarms_DB.AlarmWord_23.AlarmWord.9, bConfirm:= bConfirm);
alarms[362](evtEntry:= Tc_Events.AlarmWord23.b10, bEvt:= Alarms_DB.AlarmWord_23.AlarmWord.10, bConfirm:= bConfirm);
alarms[363](evtEntry:= Tc_Events.AlarmWord23.b11, bEvt:= Alarms_DB.AlarmWord_23.AlarmWord.11, bConfirm:= bConfirm);
alarms[364](evtEntry:= Tc_Events.AlarmWord23.b12, bEvt:= Alarms_DB.AlarmWord_23.AlarmWord.12, bConfirm:= bConfirm);
alarms[365](evtEntry:= Tc_Events.AlarmWord23.b13, bEvt:= Alarms_DB.AlarmWord_23.AlarmWord.13, bConfirm:= bConfirm);
alarms[366](evtEntry:= Tc_Events.AlarmWord23.b14, bEvt:= Alarms_DB.AlarmWord_23.AlarmWord.14, bConfirm:= bConfirm);
alarms[367](evtEntry:= Tc_Events.AlarmWord23.b15, bEvt:= Alarms_DB.AlarmWord_23.AlarmWord.15, bConfirm:= bConfirm);

//Alarm Word 24
(* uncomment when instrument is ready
Alarms_DB.AlarmWord_24.AlarmWord.0 := Trips_DB.Coil[9].ChargeRelay_FailtoClose; 
Alarms_DB.AlarmWord_24.AlarmWord.1 := Trips_DB.Coil[9].ChargeRelay_FailtoOpen;
Alarms_DB.AlarmWord_24.AlarmWord.2 := Trips_DB.Coil[10].ChargeRelay_FailtoClose;
Alarms_DB.AlarmWord_24.AlarmWord.3 := Trips_DB.Coil[10].ChargeRelay_FailtoOpen;
Alarms_DB.AlarmWord_24.AlarmWord.4 := Trips_DB.Coil[1].ACInterlockRelayFailedtoClose;
Alarms_DB.AlarmWord_24.AlarmWord.5 := Trips_DB.Coil[1].ACInterlockRelayFailedtoOpen;
Alarms_DB.AlarmWord_24.AlarmWord.6 := Trips_DB.Coil[2].ACInterlockRelayFailedtoClose;
Alarms_DB.AlarmWord_24.AlarmWord.7 := Trips_DB.Coil[2].ACInterlockRelayFailedtoOpen;
Alarms_DB.AlarmWord_24.AlarmWord.8 := Trips_DB.Coil[3].ACInterlockRelayFailedtoClose;
Alarms_DB.AlarmWord_24.AlarmWord.9 := Trips_DB.Coil[3].ACInterlockRelayFailedtoOpen;
Alarms_DB.AlarmWord_24.AlarmWord.10 := Trips_DB.Coil[4].ACInterlockRelayFailedtoClose;
Alarms_DB.AlarmWord_24.AlarmWord.11 := Trips_DB.Coil[4].ACInterlockRelayFailedtoOpen;
Alarms_DB.AlarmWord_24.AlarmWord.12 := Trips_DB.Coil[5].ACInterlockRelayFailedtoClose;
Alarms_DB.AlarmWord_24.AlarmWord.13 := Trips_DB.Coil[5].ACInterlockRelayFailedtoOpen;
Alarms_DB.AlarmWord_24.AlarmWord.14 := Trips_DB.Coil[6].ACInterlockRelayFailedtoClose;
Alarms_DB.AlarmWord_24.AlarmWord.15 := Trips_DB.Coil[6].ACInterlockRelayFailedtoOpen;
*)
//Alarm Word 24 msg
alarms[368](evtEntry:= Tc_Events.AlarmWord24.b0, bEvt:= Alarms_DB.AlarmWord_24.AlarmWord.0, bConfirm:= bConfirm);
alarms[369](evtEntry:= Tc_Events.AlarmWord24.b1, bEvt:= Alarms_DB.AlarmWord_24.AlarmWord.1, bConfirm:= bConfirm);
alarms[370](evtEntry:= Tc_Events.AlarmWord24.b2, bEvt:= Alarms_DB.AlarmWord_24.AlarmWord.2, bConfirm:= bConfirm);
alarms[371](evtEntry:= Tc_Events.AlarmWord24.b3, bEvt:= Alarms_DB.AlarmWord_24.AlarmWord.3, bConfirm:= bConfirm);
alarms[372](evtEntry:= Tc_Events.AlarmWord24.b4, bEvt:= Alarms_DB.AlarmWord_24.AlarmWord.4, bConfirm:= bConfirm);
alarms[373](evtEntry:= Tc_Events.AlarmWord24.b5, bEvt:= Alarms_DB.AlarmWord_24.AlarmWord.5, bConfirm:= bConfirm);
alarms[374](evtEntry:= Tc_Events.AlarmWord24.b6, bEvt:= Alarms_DB.AlarmWord_24.AlarmWord.6, bConfirm:= bConfirm);
alarms[375](evtEntry:= Tc_Events.AlarmWord24.b7, bEvt:= Alarms_DB.AlarmWord_24.AlarmWord.7, bConfirm:= bConfirm);
alarms[376](evtEntry:= Tc_Events.AlarmWord24.b8, bEvt:= Alarms_DB.AlarmWord_24.AlarmWord.8, bConfirm:= bConfirm);
alarms[377](evtEntry:= Tc_Events.AlarmWord24.b9, bEvt:= Alarms_DB.AlarmWord_24.AlarmWord.9, bConfirm:= bConfirm);
alarms[378](evtEntry:= Tc_Events.AlarmWord24.b10, bEvt:= Alarms_DB.AlarmWord_24.AlarmWord.10, bConfirm:= bConfirm);
alarms[379](evtEntry:= Tc_Events.AlarmWord24.b11, bEvt:= Alarms_DB.AlarmWord_24.AlarmWord.11, bConfirm:= bConfirm);
alarms[380](evtEntry:= Tc_Events.AlarmWord24.b12, bEvt:= Alarms_DB.AlarmWord_24.AlarmWord.12, bConfirm:= bConfirm);
alarms[381](evtEntry:= Tc_Events.AlarmWord24.b13, bEvt:= Alarms_DB.AlarmWord_24.AlarmWord.13, bConfirm:= bConfirm);
alarms[382](evtEntry:= Tc_Events.AlarmWord24.b14, bEvt:= Alarms_DB.AlarmWord_24.AlarmWord.14, bConfirm:= bConfirm);
alarms[383](evtEntry:= Tc_Events.AlarmWord24.b15, bEvt:= Alarms_DB.AlarmWord_24.AlarmWord.15, bConfirm:= bConfirm);

//Alarm Word 25
(* uncomment when instrument is ready
Alarms_DB.AlarmWord_25.AlarmWord.0 := Trips_DB.Coil[7].ACInterlockRelayFailedtoClose;
Alarms_DB.AlarmWord_25.AlarmWord.1 := Trips_DB.Coil[7].ACInterlockRelayFailedtoOpen;
Alarms_DB.AlarmWord_25.AlarmWord.2 := Trips_DB.Coil[8].ACInterlockRelayFailedtoClose;
Alarms_DB.AlarmWord_25.AlarmWord.3 := Trips_DB.Coil[8].ACInterlockRelayFailedtoOpen;
Alarms_DB.AlarmWord_25.AlarmWord.4 := Trips_DB.Coil[9].ACInterlockRelayFailedtoClose;
Alarms_DB.AlarmWord_25.AlarmWord.5 := Trips_DB.Coil[9].ACInterlockRelayFailedtoOpen;
Alarms_DB.AlarmWord_25.AlarmWord.6 := Trips_DB.Coil[10].ACInterlockRelayFailedtoClose;
Alarms_DB.AlarmWord_25.AlarmWord.7 := Trips_DB.Coil[10].ACInterlockRelayFailedtoOpen;
Alarms_DB.AlarmWord_25.AlarmWord.8 := Trips_DB.Coil[1].DumpRelay1_FailtoClose;
Alarms_DB.AlarmWord_25.AlarmWord.9 := Trips_DB.Coil[1].DumpRelay1_FailtoOpen;
Alarms_DB.AlarmWord_25.AlarmWord.10 := Trips_DB.Coil[2].DumpRelay1_FailtoClose;
Alarms_DB.AlarmWord_25.AlarmWord.11 := Trips_DB.Coil[2].DumpRelay1_FailtoOpen;
Alarms_DB.AlarmWord_25.AlarmWord.12 := Trips_DB.Coil[3].DumpRelay1_FailtoClose;
Alarms_DB.AlarmWord_25.AlarmWord.13 := Trips_DB.Coil[3].DumpRelay1_FailtoOpen;
Alarms_DB.AlarmWord_25.AlarmWord.14 := Trips_DB.Coil[4].DumpRelay1_FailtoClose;
Alarms_DB.AlarmWord_25.AlarmWord.15 := Trips_DB.Coil[4].DumpRelay1_FailtoOpen;
*)
//Alarm Word 25 msg
alarms[384](evtEntry:= Tc_Events.AlarmWord25.b0, bEvt:= Alarms_DB.AlarmWord_25.AlarmWord.0, bConfirm:= bConfirm);
alarms[385](evtEntry:= Tc_Events.AlarmWord25.b1, bEvt:= Alarms_DB.AlarmWord_25.AlarmWord.1, bConfirm:= bConfirm);
alarms[386](evtEntry:= Tc_Events.AlarmWord25.b2, bEvt:= Alarms_DB.AlarmWord_25.AlarmWord.2, bConfirm:= bConfirm);
alarms[387](evtEntry:= Tc_Events.AlarmWord25.b3, bEvt:= Alarms_DB.AlarmWord_25.AlarmWord.3, bConfirm:= bConfirm);
alarms[388](evtEntry:= Tc_Events.AlarmWord25.b4, bEvt:= Alarms_DB.AlarmWord_25.AlarmWord.4, bConfirm:= bConfirm);
alarms[389](evtEntry:= Tc_Events.AlarmWord25.b5, bEvt:= Alarms_DB.AlarmWord_25.AlarmWord.5, bConfirm:= bConfirm);
alarms[390](evtEntry:= Tc_Events.AlarmWord25.b6, bEvt:= Alarms_DB.AlarmWord_25.AlarmWord.6, bConfirm:= bConfirm);
alarms[391](evtEntry:= Tc_Events.AlarmWord25.b7, bEvt:= Alarms_DB.AlarmWord_25.AlarmWord.7, bConfirm:= bConfirm);
alarms[392](evtEntry:= Tc_Events.AlarmWord25.b8, bEvt:= Alarms_DB.AlarmWord_25.AlarmWord.8, bConfirm:= bConfirm);
alarms[393](evtEntry:= Tc_Events.AlarmWord25.b9, bEvt:= Alarms_DB.AlarmWord_25.AlarmWord.9, bConfirm:= bConfirm);
alarms[394](evtEntry:= Tc_Events.AlarmWord25.b10, bEvt:= Alarms_DB.AlarmWord_25.AlarmWord.10, bConfirm:= bConfirm);
alarms[395](evtEntry:= Tc_Events.AlarmWord25.b11, bEvt:= Alarms_DB.AlarmWord_25.AlarmWord.11, bConfirm:= bConfirm);
alarms[396](evtEntry:= Tc_Events.AlarmWord25.b12, bEvt:= Alarms_DB.AlarmWord_25.AlarmWord.12, bConfirm:= bConfirm);
alarms[397](evtEntry:= Tc_Events.AlarmWord25.b13, bEvt:= Alarms_DB.AlarmWord_25.AlarmWord.13, bConfirm:= bConfirm);
alarms[398](evtEntry:= Tc_Events.AlarmWord25.b14, bEvt:= Alarms_DB.AlarmWord_25.AlarmWord.14, bConfirm:= bConfirm);
alarms[399](evtEntry:= Tc_Events.AlarmWord25.b15, bEvt:= Alarms_DB.AlarmWord_25.AlarmWord.15, bConfirm:= bConfirm);

//Alarm Word 26
(* uncomment when instrument is ready
Alarms_DB.AlarmWord_26.AlarmWord.0 := Trips_DB.Coil[5].DumpRelay1_FailtoClose;
Alarms_DB.AlarmWord_26.AlarmWord.1 := Trips_DB.Coil[5].DumpRelay1_FailtoOpen;
Alarms_DB.AlarmWord_26.AlarmWord.2 := Trips_DB.Coil[6].DumpRelay1_FailtoClose;
Alarms_DB.AlarmWord_26.AlarmWord.3 := Trips_DB.Coil[6].DumpRelay1_FailtoOpen;
Alarms_DB.AlarmWord_26.AlarmWord.4 := Trips_DB.Coil[7].DumpRelay1_FailtoClose;
Alarms_DB.AlarmWord_26.AlarmWord.5 := Trips_DB.Coil[7].DumpRelay1_FailtoOpen;
Alarms_DB.AlarmWord_26.AlarmWord.6 := Trips_DB.Coil[8].DumpRelay1_FailtoClose;
Alarms_DB.AlarmWord_26.AlarmWord.7 := Trips_DB.Coil[8].DumpRelay1_FailtoOpen;
Alarms_DB.AlarmWord_26.AlarmWord.8 := Trips_DB.Coil[9].DumpRelay1_FailtoClose;
Alarms_DB.AlarmWord_26.AlarmWord.9 := Trips_DB.Coil[9].DumpRelay1_FailtoOpen;
Alarms_DB.AlarmWord_26.AlarmWord.10 := Trips_DB.Coil[10].DumpRelay1_FailtoClose;
Alarms_DB.AlarmWord_26.AlarmWord.11 := Trips_DB.Coil[10].DumpRelay1_FailtoOpen;
Alarms_DB.AlarmWord_26.AlarmWord.12 := Trips_DB.Coil[1].DumpRelay2_FailtoClose;
Alarms_DB.AlarmWord_26.AlarmWord.13 := Trips_DB.Coil[1].DumpRelay2_FailtoOpen;
Alarms_DB.AlarmWord_26.AlarmWord.14 := Trips_DB.Coil[2].DumpRelay2_FailtoClose;
Alarms_DB.AlarmWord_26.AlarmWord.15 := Trips_DB.Coil[2].DumpRelay2_FailtoOpen;
*)
//Alarm Word 26 msg
alarms[400](evtEntry:= Tc_Events.AlarmWord26.b0, bEvt:= Alarms_DB.AlarmWord_26.AlarmWord.0, bConfirm:= bConfirm);
alarms[401](evtEntry:= Tc_Events.AlarmWord26.b1, bEvt:= Alarms_DB.AlarmWord_26.AlarmWord.1, bConfirm:= bConfirm);
alarms[402](evtEntry:= Tc_Events.AlarmWord26.b2, bEvt:= Alarms_DB.AlarmWord_26.AlarmWord.2, bConfirm:= bConfirm);
alarms[403](evtEntry:= Tc_Events.AlarmWord26.b3, bEvt:= Alarms_DB.AlarmWord_26.AlarmWord.3, bConfirm:= bConfirm);
alarms[404](evtEntry:= Tc_Events.AlarmWord26.b4, bEvt:= Alarms_DB.AlarmWord_26.AlarmWord.4, bConfirm:= bConfirm);
alarms[405](evtEntry:= Tc_Events.AlarmWord26.b5, bEvt:= Alarms_DB.AlarmWord_26.AlarmWord.5, bConfirm:= bConfirm);
alarms[406](evtEntry:= Tc_Events.AlarmWord26.b6, bEvt:= Alarms_DB.AlarmWord_26.AlarmWord.6, bConfirm:= bConfirm);
alarms[407](evtEntry:= Tc_Events.AlarmWord26.b7, bEvt:= Alarms_DB.AlarmWord_26.AlarmWord.7, bConfirm:= bConfirm);
alarms[408](evtEntry:= Tc_Events.AlarmWord26.b8, bEvt:= Alarms_DB.AlarmWord_26.AlarmWord.8, bConfirm:= bConfirm);
alarms[409](evtEntry:= Tc_Events.AlarmWord26.b9, bEvt:= Alarms_DB.AlarmWord_26.AlarmWord.9, bConfirm:= bConfirm);
alarms[410](evtEntry:= Tc_Events.AlarmWord26.b10, bEvt:= Alarms_DB.AlarmWord_26.AlarmWord.10, bConfirm:= bConfirm);
alarms[411](evtEntry:= Tc_Events.AlarmWord26.b11, bEvt:= Alarms_DB.AlarmWord_26.AlarmWord.11, bConfirm:= bConfirm);
alarms[412](evtEntry:= Tc_Events.AlarmWord26.b12, bEvt:= Alarms_DB.AlarmWord_26.AlarmWord.12, bConfirm:= bConfirm);
alarms[413](evtEntry:= Tc_Events.AlarmWord26.b13, bEvt:= Alarms_DB.AlarmWord_26.AlarmWord.13, bConfirm:= bConfirm);
alarms[414](evtEntry:= Tc_Events.AlarmWord26.b14, bEvt:= Alarms_DB.AlarmWord_26.AlarmWord.14, bConfirm:= bConfirm);
alarms[415](evtEntry:= Tc_Events.AlarmWord26.b15, bEvt:= Alarms_DB.AlarmWord_26.AlarmWord.15, bConfirm:= bConfirm);

//Alarm Word 27
(* uncomment when instrument is ready
Alarms_DB.AlarmWord_27.AlarmWord.0 := Trips_DB.Coil[3].DumpRelay2_FailtoClose;
Alarms_DB.AlarmWord_27.AlarmWord.1 := Trips_DB.Coil[3].DumpRelay2_FailtoOpen;
Alarms_DB.AlarmWord_27.AlarmWord.2 := Trips_DB.Coil[4].DumpRelay2_FailtoClose;
Alarms_DB.AlarmWord_27.AlarmWord.3 := Trips_DB.Coil[4].DumpRelay2_FailtoOpen;
Alarms_DB.AlarmWord_27.AlarmWord.4 := Trips_DB.Coil[5].DumpRelay2_FailtoClose;
Alarms_DB.AlarmWord_27.AlarmWord.5 := Trips_DB.Coil[5].DumpRelay2_FailtoOpen;
Alarms_DB.AlarmWord_27.AlarmWord.6 := Trips_DB.Coil[6].DumpRelay2_FailtoClose;
Alarms_DB.AlarmWord_27.AlarmWord.7 := Trips_DB.Coil[6].DumpRelay2_FailtoOpen;
Alarms_DB.AlarmWord_27.AlarmWord.8 := Trips_DB.Coil[7].DumpRelay2_FailtoClose;
Alarms_DB.AlarmWord_27.AlarmWord.9 := Trips_DB.Coil[7].DumpRelay2_FailtoOpen;
Alarms_DB.AlarmWord_27.AlarmWord.10 := Trips_DB.Coil[8].DumpRelay2_FailtoClose;
Alarms_DB.AlarmWord_27.AlarmWord.11 := Trips_DB.Coil[8].DumpRelay2_FailtoOpen;
Alarms_DB.AlarmWord_27.AlarmWord.12:= Trips_DB.Coil[9].DumpRelay2_FailtoClose;
Alarms_DB.AlarmWord_27.AlarmWord.13 := Trips_DB.Coil[9].DumpRelay2_FailtoOpen;
Alarms_DB.AlarmWord_27.AlarmWord.14 := Trips_DB.Coil[10].DumpRelay2_FailtoClose;
Alarms_DB.AlarmWord_27.AlarmWord.15 := Trips_DB.Coil[10].DumpRelay2_FailtoOpen;
*)
//Alarm Word 27 msg
alarms[416](evtEntry:= Tc_Events.AlarmWord27.b0, bEvt:= Alarms_DB.AlarmWord_27.AlarmWord.0, bConfirm:= bConfirm);
alarms[417](evtEntry:= Tc_Events.AlarmWord27.b1, bEvt:= Alarms_DB.AlarmWord_27.AlarmWord.1, bConfirm:= bConfirm);
alarms[418](evtEntry:= Tc_Events.AlarmWord27.b2, bEvt:= Alarms_DB.AlarmWord_27.AlarmWord.2, bConfirm:= bConfirm);
alarms[419](evtEntry:= Tc_Events.AlarmWord27.b3, bEvt:= Alarms_DB.AlarmWord_27.AlarmWord.3, bConfirm:= bConfirm);
alarms[420](evtEntry:= Tc_Events.AlarmWord27.b4, bEvt:= Alarms_DB.AlarmWord_27.AlarmWord.4, bConfirm:= bConfirm);
alarms[421](evtEntry:= Tc_Events.AlarmWord27.b5, bEvt:= Alarms_DB.AlarmWord_27.AlarmWord.5, bConfirm:= bConfirm);
alarms[422](evtEntry:= Tc_Events.AlarmWord27.b6, bEvt:= Alarms_DB.AlarmWord_27.AlarmWord.6, bConfirm:= bConfirm);
alarms[423](evtEntry:= Tc_Events.AlarmWord27.b7, bEvt:= Alarms_DB.AlarmWord_27.AlarmWord.7, bConfirm:= bConfirm);
alarms[424](evtEntry:= Tc_Events.AlarmWord27.b8, bEvt:= Alarms_DB.AlarmWord_27.AlarmWord.8, bConfirm:= bConfirm);
alarms[425](evtEntry:= Tc_Events.AlarmWord27.b9, bEvt:= Alarms_DB.AlarmWord_27.AlarmWord.9, bConfirm:= bConfirm);
alarms[426](evtEntry:= Tc_Events.AlarmWord27.b10, bEvt:= Alarms_DB.AlarmWord_27.AlarmWord.10, bConfirm:= bConfirm);
alarms[427](evtEntry:= Tc_Events.AlarmWord27.b11, bEvt:= Alarms_DB.AlarmWord_27.AlarmWord.11, bConfirm:= bConfirm);
alarms[428](evtEntry:= Tc_Events.AlarmWord27.b12, bEvt:= Alarms_DB.AlarmWord_27.AlarmWord.12, bConfirm:= bConfirm);
alarms[429](evtEntry:= Tc_Events.AlarmWord27.b13, bEvt:= Alarms_DB.AlarmWord_27.AlarmWord.13, bConfirm:= bConfirm);
alarms[430](evtEntry:= Tc_Events.AlarmWord27.b14, bEvt:= Alarms_DB.AlarmWord_27.AlarmWord.14, bConfirm:= bConfirm);
alarms[431](evtEntry:= Tc_Events.AlarmWord27.b15, bEvt:= Alarms_DB.AlarmWord_27.AlarmWord.15, bConfirm:= bConfirm);
*)

//test
IF GVL.alarm_test THEN
	//i := i+1;
	Alarms_DB.MCP.AlarmWord := 16#FFFF;
	Alarms_DB.Section1.AlarmWord := 16#FFFF;
	Alarms_DB.Section2.AlarmWord := 16#FFFF;
	Alarms_DB.Section3.AlarmWord := 16#FFFF;
	Alarms_DB.Section4.AlarmWord := 16#FFFF;
	Alarms_DB.AlarmWord5.AlarmWord := 16#FFFF;
	Alarms_DB.AlarmWord7.AlarmWord := 16#FFFF;
	//Alarms_DB.Coil3.AlarmWord := 16#FFFF;
	//Alarms_DB.Coil4.AlarmWord := 16#FFFF;
	//Alarms_DB.Coil5.AlarmWord := 16#FFFF;
	//Alarms_DB.Coil6.AlarmWord := 16#FFFF;
	//Alarms_DB.Coil7.AlarmWord := 16#FFFF;
	//Alarms_DB.Coil8.AlarmWord := 16#FFFF;
	//Alarms_DB.Coil9.AlarmWord := 16#FFFF;
	//Alarms_DB.Coil10.AlarmWord := 16#FFFF;
	//Alarms_DB.AlarmWord_11.AlarmWord := 16#FFFF;
	//Alarms_DB.AlarmWord_22.AlarmWord := 16#FFFF;
	//Alarms_DB.AlarmWord_23.AlarmWord := 16#FFFF;
	//Alarms_DB.AlarmWord_24.AlarmWord := 16#FFFF;
	//Alarms_DB.AlarmWord_25.AlarmWord := 16#FFFF;
	//Alarms_DB.AlarmWord_26.AlarmWord := 16#FFFF;
	//Alarms_DB.AlarmWord_27.AlarmWord := 16#FFFF;
END_IF


//Clear Alarm Word
IF bConfirm THEN
	Alarms_DB.MCP.AlarmWord := 0;
	Alarms_DB.Section1.AlarmWord := 0;
	Alarms_DB.Section2.AlarmWord := 0;
	Alarms_DB.Section3.AlarmWord := 0;
	Alarms_DB.Section4.AlarmWord := 0;
	Alarms_DB.AlarmWord5.AlarmWord := 0;
	Alarms_DB.AlarmWord7.AlarmWord := 0;
	(*Alarms_DB.Coil3.AlarmWord := 0;
	Alarms_DB.Coil4.AlarmWord := 0;
	Alarms_DB.Coil5.AlarmWord := 0;
	Alarms_DB.Coil6.AlarmWord := 0;
	Alarms_DB.Coil7.AlarmWord := 0;
	Alarms_DB.Coil8.AlarmWord := 0;
	Alarms_DB.Coil9.AlarmWord := 0;
	Alarms_DB.Coil10.AlarmWord := 0;
	Alarms_DB.AlarmWord_11.AlarmWord := 0;
	Alarms_DB.AlarmWord_22.AlarmWord := 0;
	Alarms_DB.AlarmWord_23.AlarmWord := 0;
	Alarms_DB.AlarmWord_24.AlarmWord := 0;
	Alarms_DB.AlarmWord_25.AlarmWord := 0;
	Alarms_DB.AlarmWord_26.AlarmWord := 0;
	Alarms_DB.AlarmWord_27.AlarmWord := 0;
	*)
END_IF;

END_PROGRAM

// ---- POUs/AnalogConversion.TcPOU
PROGRAM AnalogConversion
VAR
	i					: INT := 1; //charger 1-8
	j					: INT := 1;  // section 1 - 4 
	k					: INT := 1;  // cap 1-10
	m					: INT := 1; //form cap 1-12
END_VAR

//Converting raw data into Voltage Reading (0-10V), (0.5-4.5V)   
//unfinish

//MCP Charger 
//Analog Input
//FOR i := 1 TO 8 BY 1 DO
FOR i := 1 TO 3 BY 1 DO
	
	MCP_IO.Charger[i].ChargerType_12kV := NOT MCP_IO.Charger[i].ChargerType_50kV;
	//voltage
	MCP_IO.Charger[i].voltageFeedback_norm := Norm_x (raw_input := INT_TO_REAL (MCP_IO.Charger[i].voltageFeedback_raw),
														x_max := 32767,
														x_min := 0);
	//current																									
	MCP_IO.Charger[i].currentFeedback_norm := Norm_x (raw_input := INT_TO_REAL (MCP_IO.Charger[i].currentFeedback_raw),
														x_max := 32767,
														x_min := 0);
	//50kV chargers feedback
	//if 50kV config selected
	IF MCP_IO.Charger[i].ChargerType_50kV = TRUE THEN 
		//50kv
		MCP_IO.Charger[i].voltageFeedback := (EngVal.Max_50kVChargerVoltage - EngVal.Min_50kVChargerVoltage) * ADC_10V(
																							normal_input := MCP_IO.Charger[i].voltageFeedback_norm,
																							x_max := 10,
																							x_min := 0);

		MCP_IO.Charger[i].currentFeedback := (EngVal.Max_50kVChargerCurrent - EngVal.Min_50kVChargerCurrent) * ADC_10V(
																							normal_input := MCP_IO.Charger[i].currentFeedback_norm,
																							x_max := 10,
																							x_min := 0);
		//12kv
	ELSIF MCP_IO.Charger[i].ChargerType_12kV = TRUE THEN
		MCP_IO.Charger[i].voltageFeedback := (EngVal.Max_12kVChargerVoltage - EngVal.Min_12kVChargerVoltage) * ADC_10V(
																							normal_input := MCP_IO.Charger[i].voltageFeedback_norm,
																							x_max := 10,
																							x_min := 0);
		MCP_IO.Charger[i].currentFeedback := (EngVal.Max_12kVChargerCurrent - EngVal.Min_12kVChargerCurrent) * ADC_10V(
																							normal_input := MCP_IO.Charger[i].currentFeedback_norm,
																							x_max := 10,
																							x_min := 0);										
	END_IF;	
END_FOR;

//Analog Output
//voltageSP = Required Charge Voltage******************
//limit for charing the cap
//FOR i := 1 TO 8 BY 1 DO
FOR i := 1 TO 3 BY 1 DO	
	//if 50kV config selected
	IF MCP_IO.Charger[i].ChargerType_50kV = TRUE THEN 
		//set limits of charger voltage input 
		IF MCP_IO.Charger[i].voltageSP >= REAL_TO_DINT (EngVal.UpperLimit50kVCaps) THEN
			MCP_IO.Charger[i].voltageSP := 35000; //limit at 35kV
		ELSIF MCP_IO.Charger[i].voltageSP <= 0 THEN
			MCP_IO.Charger[i].voltageSP := 0; //limit at 0V
		END_IF; 
		
	//prepare output signal for 50kV chargers.
		MCP_IO.Charger[i].voltageSP_norm := Norm_x (raw_input := DINT_TO_REAL (MCP_IO.Charger[i].voltageSP), 
												x_max := EngVal.Max_50kVChargerVoltage,
												x_min := EngVal.Min_50kVChargerVoltage);	
												
		MCP_IO.Charger[i].voltageSP_raw := AQ (norm_input := MCP_IO.Charger[i].voltageSP_norm, 
												x_max := 10,
												x_min := 0);
	END_IF;
		
	//if 12kV config selected
	IF MCP_IO.Charger[i].ChargerType_12kV = TRUE THEN
		//set limits of charger voltage input 
		IF MCP_IO.Charger[i].voltageSP <= 0 THEN
			MCP_IO.Charger[i].voltageSP := ABS(MCP_IO.Charger[i].voltageSP);
		END_IF
		
		IF MCP_IO.Charger[i].voltageSP >= REAL_TO_DINT (EngVal.UpperLimit12kVCaps) THEN
			MCP_IO.Charger[i].voltageSP := 10000; //limit at 10kV
		END_IF;

		//prepare output signal for 12kV chargers.
		MCP_IO.Charger[i].voltageSP_norm := Norm_x (raw_input := DINT_TO_REAL (MCP_IO.Charger[i].voltageSP), 
												x_max := EngVal.Max_12kVChargerVoltage,
												x_min := EngVal.Min_12kVChargerVoltage);
		
		MCP_IO.Charger[i].voltageSP_raw := AQ (norm_input := MCP_IO.Charger[i].voltageSP_norm, 
												x_max := 10,
												x_min := 0); 
	END_IF;	
												
	//limite for output sigal (<= 10V)  this should not happen
	IF MCP_IO.Charger[i].voltageSP_raw >= 32767 THEN 
		MCP_IO.Charger[i].voltageSP_raw := 32767; 										
	END_IF;
	
END_FOR;

//limits for gls 
IF MCP_IO.GLS1_voltageSP >= REAL_TO_DINT (EngVal.Max_GLS1_ChargerV) THEN 
	MCP_IO.GLS1_voltageSP := REAL_TO_DINT (EngVal.Max_GLS1_ChargerV);
	ELSIF MCP_IO.GLS1_voltageSP <= 0 THEN
		MCP_IO.GLS1_voltageSP := 0;
END_IF
IF MCP_IO.GLS2_voltageSP >= REAL_TO_DINT (EngVal.Max_GLS2_ChargerV) THEN 
	MCP_IO.GLS2_voltageSP := REAL_TO_DINT (EngVal.Max_GLS2_ChargerV);
	ELSIF MCP_IO.GLS2_voltageSP <= 0 THEN
		MCP_IO.GLS2_voltageSP := 0 ; 
END_IF
IF MCP_IO.GLS3_voltageSP >= REAL_TO_DINT (EngVal.ULimit_PreFormCapRequiredV) THEN 
	MCP_IO.GLS3_voltageSP := REAL_TO_DINT (EngVal.ULimit_PreFormCapRequiredV);
	ELSIF MCP_IO.GLS3_voltageSP <= 0 THEN
		MCP_IO.GLS3_voltageSP := 0 ; 
END_IF

//prepare analog output for gls chargers.	
MCP_IO.GLS1_voltageSP_norm := Norm_x (raw_input := DINT_TO_REAL (MCP_IO.GLS1_voltageSP),
									x_max := EngVal.Max_GLS1_ChargerV,
									x_min := 0);
MCP_IO.GLS1_voltageSP_raw:= AQ (norm_input := MCP_IO.GLS1_voltageSP_norm,
									x_max := 10,
									x_min := 0);									
									
MCP_IO.GLS2_voltageSP_norm := Norm_x (raw_input := DINT_TO_REAL (MCP_IO.GLS2_voltageSP),
									x_max := EngVal.Max_GLS2_ChargerV,
									x_min := 0);
MCP_IO.GLS2_voltageSP_raw:= AQ (norm_input := MCP_IO.GLS2_voltageSP_norm,
									x_max := 10,
									x_min := 0);	
									
MCP_IO.GLS3_voltageSP_norm := Norm_x (raw_input := DINT_TO_REAL (MCP_IO.GLS3_voltageSP),
									x_max := EngVal.Max_GLS3_ChargerV,
									x_min := 0);
MCP_IO.GLS3_voltageSP_raw:= AQ (norm_input := MCP_IO.GLS3_voltageSP_norm,
									x_max := 10,
									x_min := 0);	

//LCP 1 - 3 AI
FOR j := 1 TO 3 BY 1 DO 
	FOR k := 1 TO 10 BY 1 DO 
		LCP.Section[j].Peak.Cap[k].voltageFeedback_Norm := Norm_x (raw_input := INT_TO_REAL (LCP.Section[j].Peak.Cap[k].voltageFeedback_raw),
																x_max := 32767,
																x_min := 0);
																
		LCP.Section[j].Peak.Cap[k].voltageFeedback := (EngVal.Max_CapVoltage - EngVal.Min_CapVoltage) * ADC_10V (
																								normal_input := LCP.Section[j].Peak.Cap[k].voltageFeedback_Norm,
																								x_max := 10,
																								x_min := 0);
		//sustain caps 1 - 2
		LCP.Section[j].Sust.Cap[1].voltageFeedback_Norm := Norm_x (raw_input := INT_TO_REAL (LCP.Section[j].Sust.Cap[1].voltageFeedback_raw),
																x_max := 32767,
																x_min := 0);
																
		LCP.Section[j].Sust.Cap[1].voltageFeedback := (EngVal.Max_CapVoltage - EngVal.Min_CapVoltage) * ADC_10V (
																								normal_input := LCP.Section[j].Sust.Cap[1].voltageFeedback_Norm,
																								x_max := 10,
																								x_min := 0);
																
		LCP.Section[j].Sust.Cap[2].voltageFeedback_Norm := Norm_x (raw_input := INT_TO_REAL (LCP.Section[j].Sust.Cap[2].voltageFeedback_raw),
																x_max := 32767,
																x_min := 0);
																
		LCP.Section[j].Sust.Cap[2].voltageFeedback := (EngVal.Max_CapVoltage - EngVal.Min_CapVoltage) * ADC_10V (
																								normal_input := LCP.Section[j].Sust.Cap[2].voltageFeedback_Norm,
																								x_max := 10,
																								x_min := 0);
	END_FOR;	
END_FOR

//LCP 4 AI
FOR m := 1 TO 12 BY 1 DO
	LCP.Section[4].Form.Cap[m].voltageFeedback_norm := Norm_x (raw_input := INT_TO_REAL (LCP.Section[4].Form.Cap[m].voltageFeedback_raw),
																x_max := 32767,
																x_min := 0);
																
	LCP.Section[4].Form.Cap[m].voltageFeedback := (EngVal.Max_CapVoltage - EngVal.Min_CapVoltage) * ADC_10V (
																							normal_input := LCP.Section[4].Form.Cap[m].voltageFeedback_norm,
																							x_max := 10,
																							x_min := 0);
END_FOR;

//preform  cap AI
LCP.Section[4].PreFormCapVoltage_norm := Norm_x (raw_input := INT_TO_REAL (LCP.Section[4].PreFormCapVoltage_raw),
														x_max := 32767,
														x_min := 0);
															
LCP.Section[4].PreFormCapVoltageFeedback := (EngVal.Max_CapVoltage - EngVal.Min_CapVoltage) * ADC_10V (
																							normal_input := LCP.Section[4].PreFormCapVoltage_norm,
																							x_max := 10,
																							x_min := 0);															


//reset counter
//IF i > 8 THEN
IF i > 3 THEN
	i:=1;
END_IF;

IF j > 3 THEN 
	j := 1;
END_IF

IF k > 10 THEN 
	k := 1;
END_IF

IF m > 12 THEN 
	m := 1;
END_IF

END_PROGRAM

// ---- POUs/ChargeTime.TcPOU
PROGRAM ChargeTime
VAR

	lca_charge_cal	 : ARRAY [1..8] OF LCA_CAL;
	i				 : INT := 1; // 1-8 instances
	j				 : INT := 1; //1 - 8 ch
	m				 : INT := 1;
	
	a				 : INT := 1; 
	
	Q				 : REAL := 1; // Charge
	Current			 : REAL := 0.1; //100mA
	
	longestChargeTime: REAL;
	
END_VAR

(*IF HMI_DB.RemoteModeSelected = FALSE THEN 
	HMI_DB.TDKLoad[1].PSratedV := 12; //veto at 10
	HMI_DB.TDKLoad[2].PSratedV := 12;
	HMI_DB.TDKLoad[3].PSratedV := 12;
	HMI_DB.TDKLoad[4].PSratedV := 12;
	HMI_DB.TDKLoad[5].PSratedV := 12;
	HMI_DB.TDKLoad[6].PSratedV := 12;
	HMI_DB.TDKLoad[7].PSratedV := 50; //veto at 35
	HMI_DB.TDKLoad[8].PSratedV := 50;
	HMI_DB.GLSLoad.PSratedV := 30;
	
	HMI_DB.TDKLoad[1].TotalCapacitance := 10000;
	HMI_DB.TDKLoad[2].TotalCapacitance := 10000;
	HMI_DB.TDKLoad[3].TotalCapacitance := 10000;
	HMI_DB.TDKLoad[4].TotalCapacitance := 16000;
	HMI_DB.TDKLoad[5].TotalCapacitance := 16000;
	HMI_DB.TDKLoad[6].TotalCapacitance := 16000;
	HMI_DB.TDKLoad[7].TotalCapacitance := 1200;
	HMI_DB.TDKLoad[8].TotalCapacitance := 1200;
	HMI_DB.GLSLoad.TotalCapacitance := 200;
	
END_IF*)

IF Recipe.PeakSupplyEN = FALSE THEN
	Recipe.TDKLoad[1].RequiredChargedV :=0;
	Setpoints.TDKLoad[1].RequiredChargedV := 0;
	Recipe.TDKLoad[2].RequiredChargedV :=0;
	Setpoints.TDKLoad[2].RequiredChargedV := 0;
	Recipe.TDKLoad[3].RequiredChargedV :=0;
	Setpoints.TDKLoad[3].RequiredChargedV := 0;
END_IF

(*IF Recipe.SustSupplyEN = FALSE THEN
	Recipe.TDKLoad[4].RequiredChargedV :=0;
	Setpoints.TDKLoad[4].RequiredChargedV := 0;
	Recipe.TDKLoad[5].RequiredChargedV :=0;
	Setpoints.TDKLoad[5].RequiredChargedV := 0;
	Recipe.TDKLoad[6].RequiredChargedV :=0;
	Setpoints.TDKLoad[6].RequiredChargedV := 0;
END_IF

IF Recipe.FormSupplyEN = FALSE THEN
	Recipe.TDKLoad[7].RequiredChargedV := 0;
	Setpoints.TDKLoad[7].RequiredChargedV := 0;
	Recipe.TDKLoad[8].RequiredChargedV := 0;
	Setpoints.TDKLoad[8].RequiredChargedV := 0;
END_IF*)

IF Recipe.PFormSupplyEN = FALSE THEN
	Recipe.GLSLoad.RequiredChargedV := 0;
	Setpoints.GLSLoad.RequiredChargedV := 0;
END_IF

//veto
//this should not happen
FOR m := 1 TO 6 BY 1 DO
	IF Setpoints.TDKLoad[m].RequiredChargedV <= -2 THEN
		Setpoints.TDKLoad[m].RequiredChargedV := -2;
	END_IF	
END_FOR

IF Setpoints.GLSLoad.RequiredChargedV <= 0 THEN
	Setpoints.GLSLoad.RequiredChargedV := 0;
END_IF	

//ch 1 - 3
IF Setpoints.TDKLoad[1].RequiredChargedV >= 10 THEN
	Setpoints.TDKLoad[1].RequiredChargedV := 10;
	ELSIF Setpoints.TDKLoad[1].RequiredChargedV < 0 THEN
		Setpoints.TDKLoad[1].RequiredChargedV := ABS(Setpoints.TDKLoad[1].RequiredChargedV); 
END_IF
IF Setpoints.TDKLoad[2].RequiredChargedV >= 10 THEN
	Setpoints.TDKLoad[2].RequiredChargedV := 10;
	ELSIF Setpoints.TDKLoad[2].RequiredChargedV < 0 THEN
		Setpoints.TDKLoad[2].RequiredChargedV := ABS(Setpoints.TDKLoad[2].RequiredChargedV); 	
END_IF
IF Setpoints.TDKLoad[3].RequiredChargedV >= 10 THEN
	Setpoints.TDKLoad[3].RequiredChargedV := 10;
	ELSIF Setpoints.TDKLoad[3].RequiredChargedV < 0 THEN
		Setpoints.TDKLoad[3].RequiredChargedV := ABS(Setpoints.TDKLoad[3].RequiredChargedV); 	
END_IF
(*
//ch 4-6
IF Setpoints.TDKLoad[4].RequiredChargedV >= 12 THEN
	Setpoints.TDKLoad[4].RequiredChargedV := 12;
	ELSIF Setpoints.TDKLoad[4].RequiredChargedV < 0 THEN
		Setpoints.TDKLoad[4].RequiredChargedV := ABS(Setpoints.TDKLoad[4].RequiredChargedV); 	
END_IF
IF Setpoints.TDKLoad[5].RequiredChargedV >= 12 THEN
	Setpoints.TDKLoad[5].RequiredChargedV := 12;
	ELSIF Setpoints.TDKLoad[5].RequiredChargedV < 0 THEN
		Setpoints.TDKLoad[5].RequiredChargedV := ABS(Setpoints.TDKLoad[5].RequiredChargedV); 	
END_IF
IF Setpoints.TDKLoad[6].RequiredChargedV >= 12 THEN
	Setpoints.TDKLoad[6].RequiredChargedV := 12;
	ELSIF Setpoints.TDKLoad[6].RequiredChargedV < 0 THEN
		Setpoints.TDKLoad[6].RequiredChargedV := ABS(Setpoints.TDKLoad[6].RequiredChargedV); 	
END_IF
//ch 7 - 8
IF Setpoints.TDKLoad[7].RequiredChargedV >= 35 THEN
	Setpoints.TDKLoad[7].RequiredChargedV := 35;
	ELSIF Setpoints.TDKLoad[7].RequiredChargedV <= 0  THEN
		Setpoints.TDKLoad[7].RequiredChargedV := 0; 	
END_IF
IF Setpoints.TDKLoad[8].RequiredChargedV >= 35 THEN
	Setpoints.TDKLoad[8].RequiredChargedV := 35;
	ELSIF Setpoints.TDKLoad[8].RequiredChargedV <= 0 THEN
		Setpoints.TDKLoad[8].RequiredChargedV := ABS(Setpoints.TDKLoad[8].RequiredChargedV); 	
END_IF
*)
IF Setpoints.GLSLoad.RequiredChargedV >= 30 THEN
	Setpoints.GLSLoad.RequiredChargedV := 30;
	ELSIF Setpoints.GLSLoad.RequiredChargedV <= 0 THEN
		Setpoints.GLSLoad.RequiredChargedV := 0; 	
END_IF

//mapping hmi input to setpoints
FOR j := 1 TO 8 BY 1 DO	
	Setpoints.TDKLoad[j].TotalCapacitance	:= HMI_DB.TDKLoad[j].TotalCapacitance;
	Setpoints.TDKLoad[j].PSratedV 			:= HMI_DB.TDKLoad[j].PSratedV;
	//Setpoints.PeakBank[m].RequiredChargedV	:= Recipe.PeakBank[m].RequiredChargedV; //only thing that comes from the main plc recipe
	Setpoints.TDKLoad[j].wLCA				:= HMI_DB.TDKLoad[j].wLCA;
	Setpoints.TDKLoad[j].NumOfCharger		:= HMI_DB.TDKLoad[j].NumOfCharger;	
	
	Setpoints.TDKLoad[j].TotalCapacitance	:= HMI_DB.TDKLoad[j].TotalCapacitance;
	Setpoints.TDKLoad[j].PSratedV 			:= HMI_DB.TDKLoad[j].PSratedV;
	//Setpoints.SustBank[m].RequiredChargedV	:= Recipe.SustBank[m].RequiredChargedV; //only thing that comes from the main plc recipe
	Setpoints.TDKLoad[j].wLCA				:= HMI_DB.TDKLoad[j].wLCA;
	Setpoints.TDKLoad[j].NumOfCharger		:= HMI_DB.TDKLoad[j].NumOfCharger;	
	//charge time delay and elapse for HMI
	ChargeTime_DB.ChargeTimeStartDelay[j] := TIME_TO_INT((ChargeTime_DB.ChargerDelay_PT[j] - ChargeTime_DB.ChargerDelay_ET[j])/1000);
	ChargeTime_DB.ChargingTimeElapse[j] := TIME_TO_INT((ChargeTime_DB.ChargingTimeElapse_TON[j].PT - ChargeTime_DB.ChargingTimeElapse_TON[j].ET)/1000);
END_FOR

ChargeTime_DB.PreFormChargeTimeStartDelay := TIME_TO_INT((ChargeTime_DB.PreFormChargeTime_PT - ChargeTime_DB.PreFormChargeTime_ET)/1000);
ChargeTime_DB.PreFormChargingTimeElapse := TIME_TO_INT((ChargeTime_DB.PreFormChargingTimeElapse_TON.PT - ChargeTime_DB.PreFormChargingTimeElapse_TON.ET)/1000);

//GLS 3
Setpoints.GLSLoad.TotalCapacitance	:= HMI_DB.GLSLoad.TotalCapacitance;
Setpoints.GLSLoad.PSratedV 			:= HMI_DB.GLSLoad.PSratedV;
//Setpoints.PreFormBank.RequiredChargedV	:= Recipe.PreFormBank.RequiredChargedV; //only thing that comes from the main plc recipe
//Setpoints.GLSLoad.wLCA				:= HMI_DB.GLSLoad.wLCA;
Setpoints.GLSLoad.NumOfCharger		:= HMI_DB.GLSLoad.NumOfCharger;	

//chg time
//FOR i := 1 TO 8 BY 1 DO
FOR i := 1 TO 3 BY 1 DO
	lca_charge_cal[i](	PSratedV := Setpoints.TDKLoad[i].PSratedV, 
						RequiredChargeV := Setpoints.TDKLoad[i].RequiredChargedV, 
						LoadCapacitance := Setpoints.TDKLoad[i].TotalCapacitance, 
						NumOfCharger := Setpoints.TDKLoad[i].NumOfCharger, 
						wLCA := Setpoints.TDKLoad[i].wLCA
						);

	MCP_IO.Charger[i].ChargeTime.timeToChargeLoad := lca_charge_cal[i].TimeToChargeLoad;
	MCP_IO.Charger[i].ChargeTime.Power := lca_charge_cal[i].RespectedPower;
END_FOR


//gls - gls3 is preform cap charger
Q := 1000* Setpoints.GLSLoad.RequiredChargedV * (Setpoints.GLSLoad.TotalCapacitance / 1000000);
MCP_IO.GLS3_Load.timeToChargeLoad := Q / Current;
MCP_IO.GLS3_Load.Power := 1000*Setpoints.GLSLoad.RequiredChargedV * Current;

//find the longest charge time.  //need more work
longestChargeTime := MAX( MCP_IO.Charger[1].ChargeTime.timeToChargeLoad,
							MCP_IO.Charger[2].ChargeTime.timeToChargeLoad,
							MCP_IO.Charger[3].ChargeTime.timeToChargeLoad,
							(*MCP_IO.Charger[4].ChargeTime.timeToChargeLoad,
							MCP_IO.Charger[5].ChargeTime.timeToChargeLoad,
							MCP_IO.Charger[6].ChargeTime.timeToChargeLoad,
							MCP_IO.Charger[7].ChargeTime.timeToChargeLoad,
							MCP_IO.Charger[8].ChargeTime.timeToChargeLoad, *)
							MCP_IO.GLS3_Load.timeToChargeLoad);

ChargeTime_DB.LongestChargeTime_PT := REAL_TO_TIME (1000*longestChargeTime);

//FOR a := 1 TO 8 BY 1 DO
FOR a := 1 TO 3 BY 1 DO
	IF (longestChargeTime - MCP_IO.Charger[a].ChargeTime.timeToChargeLoad) >= 0 THEN
		ChargeTime_DB.ChargerDelay_PT[a] := REAL_TO_TIME (1000*(longestChargeTime - MCP_IO.Charger[a].ChargeTime.timeToChargeLoad));
		ELSE 
			ChargeTime_DB.ChargerDelay_PT[a] := REAL_TO_TIME (1000*(MCP_IO.Charger[a].ChargeTime.timeToChargeLoad - longestChargeTime));
	END_IF;		
		
	//IF (longestChargeTime - MCP_IO.Charger[a+3].ChargeTime.timeToChargeLoad) >= 0 THEN
	//	ChargeTime_DB.SustChargeTime_PT[a] := REAL_TO_TIME (1000*(longestChargeTime - MCP_IO.Charger[a+3].ChargeTime.timeToChargeLoad));	
	//END_IF;	
	
END_FOR;


(*IF (longestChargeTime - MCP_IO.Charger[7].ChargeTime.timeToChargeLoad) >= 0 THEN
	ChargeTime_DB.FormChargeTime_PT[1] := REAL_TO_TIME (1000*(longestChargeTime - MCP_IO.Charger[7].ChargeTime.timeToChargeLoad));	
END_IF;	
IF (longestChargeTime - MCP_IO.Charger[8].ChargeTime.timeToChargeLoad) >= 0 THEN
	ChargeTime_DB.FormChargeTime_PT[2] := REAL_TO_TIME (1000*(longestChargeTime - MCP_IO.Charger[8].ChargeTime.timeToChargeLoad));	
END_IF;	
*)
IF (longestChargeTime - MCP_IO.GLS3_Load.timeToChargeLoad) >= 0 THEN
		ChargeTime_DB.PreFormChargeTime_PT := REAL_TO_TIME (1000*(longestChargeTime - MCP_IO.GLS3_Load.timeToChargeLoad));
		ELSE
			ChargeTime_DB.PreFormChargeTime_PT := REAL_TO_TIME (1000*(MCP_IO.GLS3_Load.timeToChargeLoad -longestChargeTime));
END_IF;



//IF i > 8 THEN 
IF i > 3 THEN 
	i := 0;
END_IF

IF j > 8 THEN
	j := 0;
END_IF

IF m > 6 THEN
	m := 0;
END_IF

//IF a > 8 THEN
IF a > 3 THEN
	a := 1;
END_IF;

END_PROGRAM

// ---- POUs/Dump_FB.TcPOU
FUNCTION_BLOCK Dump_FB
VAR_INPUT
	EN : BOOL;
	IN1 : BOOL; //AllCapsDischarged
	IN2 : BOOL; //AllDumpRelaysOpen
	//IN3 : BOOL; //DumpingRunOut	 
	//Heartbeat		  : BOOL;
END_VAR
VAR_OUTPUT
	DONE : BOOL;
	DumpingRunOut_Elapse : REAL;
END_VAR
VAR
	//AbortPSnRlyDelayDONE : BOOL;
	//AbortPSnRlyDelay_Timer : TON;
	//AbortPSnRlyDelay_PT : TIME;
	DumpingRunOutTMR_TON : TON;
	DumpingRunOutTMR_PT : TIME := T#190S;
	DumpingRunOutTMR_ET : TIME;
	
	i : USINT := 1;
	j : USINT := 1;
	k : USINT := 0;
END_VAR


IF EN = TRUE THEN
	//start dump runout timer
	DumpingRunOutTMR_TON (IN := TRUE, PT := DumpingRunOutTMR_PT, ET => DumpingRunOutTMR_ET);
	DumpingRunOut_Elapse := TIME_TO_REAL((DumpingRunOutTMR_PT - DumpingRunOutTMR_ET)/1000);
	//IF DumpingRunOut = TRUE AND AllCapsDischarged = TRUE AND AllDumpRelaysOpen = FALSE THEN 
	//	DONE := TRUE;
	//	ELSE 
	//		DONE := FALSE;
	//END_IF
		//	DONE := TRUE;
	//IF Heartbeat = TRUE THEN 
	//	 k := k + 1;
	//END_IF;			
	IF DumpingRunOutTMR_TON.Q = TRUE AND Permissives_DB.AllSectCapsDischarged = TRUE AND IN2 = TRUE THEN //if timer run out, and in remoter mode go to trip
		DONE := TRUE;
		DumpingRunOutTMR_TON (IN := FALSE);
		ELSE 
			DONE := FALSE; 
	END_IF
					
	//TURN OFF ALL CHARGERS
	//FOR i := 1 TO 8 BY 1 DO 
	FOR i := 1 TO 3 BY 1 DO
		MCP_IO.Charger[i].inhibit := TRUE; 		
		MCP_IO.Charger[i].HV_ON := FALSE; 
		MCP_IO.Charger[i].voltageSP := 0;
			
		//ChargeTime_DB.ChargingTimeElapse_TON[i] (IN := FALSE); //reset charging time elapse
	END_FOR;

	MCP_IO.GLS1_hvON := FALSE;
	MCP_IO.GLS2_hvON := FALSE;
	MCP_IO.GLS3_hvON := FALSE;
	MCP_IO.GLS1_voltageSP := 0;
	MCP_IO.GLS2_voltageSP := 0;
	MCP_IO.GLS3_voltageSP := 0;
					
	//ChargeTime_DB.PreFormChargingTimeElapse_TON (IN := FALSE);
	//start delay
	//AbortPSnRlyDelay_Timer (IN := TRUE, PT := AbortPSnRlyDelay_PT);					
					
	//IF AbortPSnRlyDelay_Timer.Q = TRUE THEN 
	//	AbortPSnRlyDelayDONE := TRUE;
	//	AbortPSnRlyDelay_Timer (IN := FALSE);
	//END_IF;
					
//IF 	AbortPSnRlyDelayDONE = TRUE THEN
	FOR j := 1 TO 3 BY 1 DO 
		//Open all charge relays
		LCP.Section[j].Peak.CloseChargeRelay1 := FALSE; 
		LCP.Section[j].Peak.CloseChargeRelay2 := FALSE; 
		LCP.Section[j].Sust.CloseChargeRelay1 := FALSE;
		LCP.Section[j].Sust.CloseChargeRelay2 := FALSE;
		//close all dump relays  - for SAFE STATE they can all go together
		LCP.Section[j].Peak.OpenDumpRelay1 := FALSE;
		LCP.Section[j].Peak.OpenDumpRelay2 := FALSE;
		LCP.Section[j].Sust.OpenDumpRelay1 := FALSE;
		LCP.Section[j].Sust.OpenDumpRelay2 := FALSE;	
	END_FOR;
	//open all charge rly on form
	LCP.Section[4].Form.CloseChargeRelay1 := FALSE;
	LCP.Section[4].Form.CloseChargeRelay2 := FALSE;
	LCP.Section[4].Form.CloseFormTrigChargeRly := FALSE;
	LCP.Section[4].Form.ClosePreFormChargeRly := FALSE;
	LCP.Section[4].Form.ClosePreFormTrigChargeRly := FALSE;
	//close all dump relay on form
	LCP.Section[4].Form.OpenDumpRelay1 := FALSE;
	LCP.Section[4].Form.OpenDumpRelay2 := FALSE;
	LCP.Section[4].Form.OpenPreFormDumpRly := FALSE;
	LCP.Section[4].Form.OpenFormTrigDumpRly1 := FALSE;
	LCP.Section[4].Form.OpenPreFormTrigDumpRly1 := FALSE;
						
	//AbortPSnRlyDelay_Timer (IN := FALSE);
	//AbortPSnRlyDelayDONE := FALSE;
ELSE
	DumpingRunOutTMR_TON (IN := FALSE);
END_IF;
					
//IF i > 8 THEN
IF i > 3 THEN
	i := 1;
END_IF
					
IF j > 3 THEN
	j := 1;
END_IF

END_FUNCTION_BLOCK

// ---- POUs/HMI.TcPOU
PROGRAM HMI
VAR
END_VAR

IF MCP_IO.RemoteModeSelected = TRUE OR HMI_DB.RemoteModeSelected = TRUE THEN 
	GVL.RemoteModeSelected := TRUE;
ELSIF MCP_IO.RemoteModeSelected = FALSE OR HMI_DB.RemoteModeSelected = FALSE THEN
		GVL.RemoteModeSelected := FALSE;
END_IF

END_PROGRAM

// ---- POUs/MAIN.TcPOU
PROGRAM MAIN
VAR
END_VAR

Alias();
Heartbeat();
Permissives();
Trips();
Alarms();
Sequence();
Communication();
Analogconversion();
HMI();
ChargeTime();

END_PROGRAM

// ---- POUs/Permissives.TcPOU
PROGRAM Permissives
VAR
	i : INT := 1;  //for section 1 - 3 
	j : INT := 1; //for charger 1-8
	k : INT := 1; //cap 1- 10
	m : INT := 1; //form cap 1-12
	n : INT := 1; //1-6
	p : INT := 7; //7-12
END_VAR

//Charger summary faults
//Trips_DB.AnySummaryFault = FALSE AND Trips_DB.AnyEstopPressed //add to no fault detected.

//section ready to charge
FOR i := 1 TO 3 BY 1 DO
	IF Trips_DB.NoFaultDetected = TRUE AND //MCP_IO.Charger[1-8].HVisOn AND
		Permissives_DB.AllChargeRelaysClosed = TRUE AND
		LCP.Section[i].Peak.ShortContact1Engaged = FALSE AND
		LCP.Section[i].Peak.ShortContact2Engaged = FALSE AND
		LCP.Section[i].Sust.ShortContact1Engaged = FALSE AND
		LCP.Section[i].Sust.ShortContact2Engaged = FALSE
	THEN
		LCP.Section[i].SystemReadyToCharge := TRUE;	
	ELSE
		LCP.Section[i].SystemReadyToCharge := FALSE;		
	END_IF;
END_FOR;

//Section 4
IF Trips_DB.NoFaultDetected = TRUE AND //MCP_IO.Charger[1-8].HVisOn AND
	Permissives_DB.AllChargeRelaysClosed = TRUE AND
	LCP.Section[4].Form.ShortContact1Engaged = FALSE AND
	LCP.Section[4].Form.ShortContact2Engaged = FALSE AND
	LCP.Section[4].Form.FormTrigShortContactEngaged = FALSE AND
	LCP.Section[4].Form.PreFormTrigShortContactEngaged = FALSE 
	THEN
		LCP.Section[4].SystemReadyToCharge := TRUE;
	ELSE
		LCP.Section[4].SystemReadyToCharge := FALSE;
END_IF;
	
IF LCP.Section[1].SystemReadyToCharge = TRUE AND 
	LCP.Section[2].SystemReadyToCharge = TRUE AND
	LCP.Section[3].SystemReadyToCharge = TRUE AND
	LCP.Section[4].SystemReadyToCharge = TRUE
	THEN
		Permissives_DB.AllSystemsReadytoCharge := TRUE;
		ELSE
			Permissives_DB.AllSystemsReadytoCharge := FALSE;
END_IF


// shorts and unshorts
//Peaking  -- short contacts are NO, so if close is false, it is and unshort is true, then it is not shorted 
FOR i := 1 TO 3 BY 1 DO
	IF LCP.Section[i].Peak.ShortContact1_close = TRUE AND LCP.Section[i].Peak.UnshortContact1_close = FALSE 
		THEN
			LCP.Section[i].Peak.ShortContact1Engaged := TRUE;
		ELSE
			LCP.Section[i].Peak.ShortContact1Engaged := FALSE;
	END_IF;
	
	IF LCP.Section[i].Peak.ShortContact2_close = TRUE AND LCP.Section[i].Peak.UnshortContact2_close = FALSE 
		THEN
			LCP.Section[i].Peak.ShortContact2Engaged := TRUE;
		ELSE
			LCP.Section[i].Peak.ShortContact2Engaged := FALSE;
	END_IF;
	
END_FOR;

//Sustain
FOR i := 1 TO 3 BY 1 DO
	IF LCP.Section[i].Sust.ShortContact1_close = TRUE AND LCP.Section[i].Sust.UnshortContact1_close = FALSE 
		THEN
			LCP.Section[i].Sust.ShortContact1Engaged := TRUE;
		ELSE
			LCP.Section[i].Sust.ShortContact1Engaged := FALSE;
	END_IF;
	
	IF LCP.Section[i].Sust.ShortContact2_close = TRUE AND LCP.Section[i].Sust.UnshortContact2_close = FALSE 
		THEN
			LCP.Section[i].Sust.ShortContact2Engaged := TRUE;
		ELSE
			LCP.Section[i].Sust.ShortContact2Engaged := FALSE;
	END_IF;
	
END_FOR;

//Formation
IF LCP.Section[4].Form.ShortContact1_close = TRUE AND LCP.Section[4].Form.UnshortContact1_close = FALSE
	THEN
		LCP.Section[4].Form.ShortContact1Engaged := TRUE;
	ELSE
		LCP.Section[4].Form.ShortContact1Engaged := FALSE; //might need to clarify on the NC of the short contacts.
END_IF;

IF LCP.Section[4].Form.ShortContact2_close = TRUE AND LCP.Section[4].Form.UnshortContact2_close = FALSE 
	THEN
		LCP.Section[4].Form.ShortContact2Engaged := TRUE;
	ELSE
		LCP.Section[4].Form.ShortContact2Engaged := FALSE; //might need to clarify on the NC of the short contacts.
END_IF;

// form trig short 
IF LCP.Section[4].Form.FormTrigShortContact_close = TRUE AND LCP.Section[4].Form.FormTrigUnShortContact_close = FALSE
	THEN
		LCP.Section[4].Form.FormTrigShortContactEngaged := TRUE;
	ELSE
		LCP.Section[4].Form.FormTrigShortContactEngaged := FALSE;
END_IF
// preform trig short 
IF LCP.Section[4].Form.PreFormTrigShortContact_close = TRUE AND LCP.Section[4].Form.PreFormTrigUnShortContact_close = FALSE
	THEN
		LCP.Section[4].Form.PreFormTrigShortContactEngaged := TRUE;
	ELSE
		LCP.Section[4].Form.PreFormTrigShortContactEngaged := FALSE;
END_IF

//short contacts unknown - This should have never happen
FOR i := 1 TO 3 BY 1 DO
	//Peak
	IF (LCP.Section[i].Peak.ShortContact1_close = TRUE AND LCP.Section[i].Peak.UnShortContact1_close = TRUE) OR 
 		(LCP.Section[i].Peak.ShortContact1_close = FALSE AND LCP.Section[i].Peak.UnShortContact1_close = FALSE)
		THEN
			LCP.Section[i].Peak.ShortContact1unknown := TRUE;
			ELSE
				LCP.Section[i].Peak.ShortContact1unknown := FALSE;
	END_IF;
	
	IF (LCP.Section[i].Peak.ShortContact2_close = TRUE AND LCP.Section[i].Peak.UnShortContact2_close = TRUE) OR 
 		(LCP.Section[i].Peak.ShortContact2_close = FALSE AND LCP.Section[i].Peak.UnShortContact2_close = FALSE)
		THEN
			LCP.Section[i].Peak.ShortContact2unknown := TRUE;
			ELSE
				LCP.Section[i].Peak.ShortContact2unknown := FALSE;
	END_IF;
	//Sust
	IF (LCP.Section[i].Sust.ShortContact1_close = TRUE AND LCP.Section[i].Sust.UnShortContact1_close = TRUE) OR 
 		(LCP.Section[i].Sust.ShortContact1_close = FALSE AND LCP.Section[i].Sust.UnShortContact1_close = FALSE)
		THEN
			LCP.Section[i].Sust.ShortContact1unknown := TRUE;
			ELSE
				LCP.Section[i].Sust.ShortContact1unknown := FALSE;
	END_IF;	
	
	IF (LCP.Section[i].Sust.ShortContact2_close = TRUE AND LCP.Section[i].Sust.UnShortContact2_close = TRUE) OR 
 		(LCP.Section[i].Sust.ShortContact2_close = FALSE AND LCP.Section[i].Sust.UnShortContact2_close = FALSE)
		THEN
			LCP.Section[i].Sust.ShortContact2unknown := TRUE;
			ELSE
				LCP.Section[i].Sust.ShortContact2unknown := FALSE;
	END_IF;	
	
END_FOR;

//Formation
IF (LCP.Section[4].Form.ShortContact1_close = TRUE AND LCP.Section[4].Form.UnShortContact1_close = TRUE) OR 
 	(LCP.Section[4].Form.ShortContact1_close = FALSE AND LCP.Section[4].Form.UnShortContact1_close = FALSE)
	THEN
		LCP.Section[4].Form.ShortContact1unknown := TRUE;
		ELSE
			LCP.Section[4].Form.ShortContact1unknown := FALSE;
END_IF;	
	
IF (LCP.Section[4].Form.ShortContact2_close = TRUE AND LCP.Section[4].Form.UnShortContact2_close = TRUE) OR 
 	(LCP.Section[4].Form.ShortContact2_close = FALSE AND LCP.Section[4].Form.UnShortContact2_close = FALSE)
	THEN
		LCP.Section[4].Form.ShortContact2unknown := TRUE;
		ELSE
			LCP.Section[4].Form.ShortContact2unknown := FALSE;
END_IF;	

IF (LCP.Section[4].Form.FormTrigUnshortContact_close = TRUE AND LCP.Section[4].Form.FormTrigUnshortContact_close = TRUE) OR 
	(LCP.Section[4].Form.FormTrigUnshortContact_close = FALSE AND LCP.Section[4].Form.FormTrigUnshortContact_close = FALSE)
	THEN 
		LCP.Section[4].Form.FormTrigShortContactUnknown := TRUE;
		ELSE
			LCP.Section[4].Form.FormTrigShortContactUnknown := FALSE;
END_IF;

IF (LCP.Section[4].Form.PreFormTrigShortContact_close = TRUE AND LCP.Section[4].Form.PreFormTrigUnShortContact_close = TRUE) OR
	(LCP.Section[4].Form.PreFormTrigShortContact_close = FALSE AND LCP.Section[4].Form.PreFormTrigUnShortContact_close = FALSE)
	THEN
		LCP.Section[4].Form.PreFormTrigShortContactUnknown := TRUE;
		ELSE
			LCP.Section[4].Form.PreFormTrigShortContactUnknown := FALSE;
END_IF;
	
// any short contact in unknown state?
IF LCP.Section[1].Peak.ShortContact1unknown = FALSE AND 
	LCP.Section[1].Peak.ShortContact2unknown = FALSE AND
	LCP.Section[2].Peak.ShortContact1unknown = FALSE AND
	LCP.Section[2].Peak.ShortContact2unknown = FALSE AND
	LCP.Section[3].Peak.ShortContact1unknown = FALSE AND
	LCP.Section[3].Peak.ShortContact2unknown = FALSE AND
	LCP.Section[1].Sust.ShortContact1unknown = FALSE AND
	LCP.Section[1].Sust.ShortContact2unknown = FALSE AND
	LCP.Section[2].Sust.ShortContact1unknown = FALSE AND 
	LCP.Section[2].Sust.ShortContact2unknown = FALSE AND
	LCP.Section[3].Sust.ShortContact1unknown = FALSE AND 
	LCP.Section[3].Sust.ShortContact2unknown = FALSE AND
	LCP.Section[4].Form.ShortContact1unknown = FALSE AND
	LCP.Section[4].Form.ShortContact2unknown = FALSE AND 
	LCP.Section[4].Form.FormTrigShortContactUnknown = FALSE AND //
	LCP.Section[4].Form.PreFormTrigShortContactUnknown = FALSE //
	THEN
		Permissives_DB.NoShortingUnknowns := TRUE;
	ELSE
		Permissives_DB.NoShortingUnknowns := FALSE;
END_IF;


//any short contact engaged

IF LCP.Section[1].Peak.ShortContact1Engaged = TRUE AND 
	LCP.Section[1].Peak.ShortContact2Engaged = TRUE AND
	LCP.Section[2].Peak.ShortContact1Engaged = TRUE AND
	LCP.Section[2].Peak.ShortContact2Engaged = TRUE AND
	LCP.Section[3].Peak.ShortContact1Engaged = TRUE AND
	LCP.Section[3].Peak.ShortContact2Engaged = TRUE AND
	LCP.Section[1].Sust.ShortContact1Engaged = TRUE AND
	LCP.Section[1].Sust.ShortContact2Engaged = TRUE AND
	LCP.Section[2].Sust.ShortContact1Engaged = TRUE AND 
	LCP.Section[2].Sust.ShortContact2Engaged = TRUE AND
	LCP.Section[3].Sust.ShortContact1Engaged = TRUE AND 
	LCP.Section[3].Sust.ShortContact2Engaged = TRUE AND
	LCP.Section[4].Form.ShortContact1Engaged = TRUE AND
	LCP.Section[4].Form.ShortContact2Engaged = TRUE AND 
	LCP.Section[4].Form.FormTrigShortContactEngaged = TRUE AND //
	LCP.Section[4].Form.PreFormTrigShortContactEngaged = TRUE //
	THEN
		Permissives_DB.AllShortContactEngaged := TRUE;
	ELSE 
		Permissives_DB.AllShortContactEngaged := FALSE;	
END_IF;

//All charger inhibited
IF (MCP_IO.Charger[1].inhibited = TRUE OR Recipe.PeakSupplyEN = FALSE) AND
	(MCP_IO.Charger[2].inhibited = TRUE OR Recipe.PeakSupplyEN = FALSE) AND
	(MCP_IO.Charger[3].inhibited = TRUE OR Recipe.PeakSupplyEN = FALSE) //AND
	//(MCP_IO.Charger[4].inhibited = TRUE OR Recipe.SustSupplyEN = FALSE) AND
	//(MCP_IO.Charger[5].inhibited = TRUE OR Recipe.SustSupplyEN = FALSE) AND
	//(MCP_IO.Charger[6].inhibited = TRUE OR Recipe.SustSupplyEN = FALSE) AND
	//(MCP_IO.Charger[7].inhibited = TRUE OR Recipe.FormSupplyEN = FALSE) AND
	//(MCP_IO.Charger[8].inhibited = TRUE OR Recipe.FormSupplyEN = FALSE) 
	THEN
		Permissives_DB.AllChargerInhibited := TRUE;
		ELSE
			Permissives_DB.AllChargerInhibited := FALSE;
END_IF;

//All charger HV ON
IF (MCP_IO.Charger[1].HV_isON = TRUE OR Recipe.PeakSupplyEN = FALSE) AND
	(MCP_IO.Charger[2].HV_isON = TRUE OR Recipe.PeakSupplyEN = FALSE) AND
	(MCP_IO.Charger[3].HV_isON = TRUE OR Recipe.PeakSupplyEN = FALSE) (*AND
	(MCP_IO.Charger[4].HV_isON = TRUE OR Recipe.SustSupplyEN = FALSE) AND
	(MCP_IO.Charger[5].HV_isON = TRUE OR Recipe.SustSupplyEN = FALSE) AND
	(MCP_IO.Charger[6].HV_isON = TRUE OR Recipe.SustSupplyEN = FALSE) AND
	(MCP_IO.Charger[7].HV_isON = TRUE OR Recipe.FormSupplyEN = FALSE) AND
	(MCP_IO.Charger[8].HV_isON = TRUE OR Recipe.FormSupplyEN = FALSE) AND
	(MCP_IO.GLS3_hvON = TRUE OR Recipe.PFormSupplyEN = FALSE)*)
	THEN
		Permissives_DB.AllChargerHVisON := TRUE;
		ELSE
			Permissives_DB.AllChargerHVisON := FALSE;
END_IF;

//peaking ch hv on
IF MCP_IO.Charger[1].HV_isON = TRUE AND 
	MCP_IO.Charger[2].HV_isON = TRUE AND 
	MCP_IO.Charger[3].HV_isON = TRUE 
	THEN
		Permissives_DB.AllPeakChargerHVisON := TRUE;
		ELSE
			Permissives_DB.AllPeakChargerHVisON := FALSE;
END_IF
//sustain ch hv on
(*IF MCP_IO.Charger[4].HV_isON = TRUE AND 
	MCP_IO.Charger[5].HV_isON = TRUE AND 
	MCP_IO.Charger[6].HV_isON = TRUE 
	THEN
		Permissives_DB.AllSustChargerHVisON := TRUE;
		ELSE
			Permissives_DB.AllSustChargerHVisON := FALSE;
END_IF
//Form ch hv on
IF MCP_IO.Charger[7].HV_isON = TRUE AND 
	MCP_IO.Charger[8].HV_isON = TRUE  
	THEN
		Permissives_DB.AllFormChargerHVisON := TRUE;
		ELSE
			Permissives_DB.AllFormChargerHVisON := FALSE;
END_IF*)
//peaking ch inhibit
IF MCP_IO.Charger[1].inhibited = TRUE AND 
	MCP_IO.Charger[2].inhibited = TRUE AND 
	MCP_IO.Charger[3].inhibited = TRUE 
	THEN
		Permissives_DB.AllPeakChargerInhibited := TRUE;
		ELSE
			Permissives_DB.AllPeakChargerInhibited := FALSE;
END_IF
//sust ch inhibit
(*IF MCP_IO.Charger[4].inhibited = TRUE AND 
	MCP_IO.Charger[5].inhibited = TRUE AND 
	MCP_IO.Charger[6].inhibited = TRUE 
	THEN
		Permissives_DB.AllSustChargerInhibited := TRUE;
		ELSE
			Permissives_DB.AllSustChargerInhibited := FALSE;
END_IF
//form ch inhibit
IF MCP_IO.Charger[7].inhibited = TRUE AND 
	MCP_IO.Charger[8].inhibited = TRUE
	THEN
		Permissives_DB.AllFormChargerInhibited := TRUE;
		ELSE
			Permissives_DB.AllFormChargerInhibited := FALSE;
END_IF*)

IF (MCP_IO.Charger[1].EndOfCharge = TRUE OR Recipe.PeakSupplyEN = FALSE) AND
	(MCP_IO.Charger[2].EndOfCharge = TRUE OR Recipe.PeakSupplyEN = FALSE) AND
	(MCP_IO.Charger[3].EndOfCharge = TRUE OR Recipe.PeakSupplyEN = FALSE) (*AND
	(MCP_IO.Charger[4].EndOfCharge = TRUE OR Recipe.SustsupplyEN = FALSE) AND
	(MCP_IO.Charger[5].EndOfCharge = TRUE OR Recipe.SustsupplyEN = FALSE) AND
	(MCP_IO.Charger[6].EndOfCharge = TRUE OR Recipe.SustsupplyEN = FALSE) AND
	(MCP_IO.Charger[7].EndOfCharge = TRUE OR Recipe.FormSupplyEN = FALSE) AND
	(MCP_IO.Charger[8].EndOfCharge = TRUE OR Recipe.FormSupplyEN = FALSE) *)
	THEN 
		Permissives_DB.AllChargerEOC := TRUE;
		ELSE
			Permissives_DB.AllChargerEOC := FALSE;
END_IF

//all peaking charg
IF LCP.Section[1].Peak.ChargeRelay1_close = TRUE AND
	LCP.Section[1].Peak.ChargeRelay2_close = TRUE AND
	LCP.Section[2].Peak.ChargeRelay1_close = TRUE AND
	LCP.Section[2].Peak.ChargeRelay2_close = TRUE AND
	LCP.Section[3].Peak.ChargeRelay1_close = TRUE AND
	LCP.Section[3].Peak.ChargeRelay2_close = TRUE 
	THEN
		Permissives_DB.AllPeakChargeRlyClose := TRUE;
		ELSE
			Permissives_DB.AllPeakChargeRlyClose := FALSE;
END_IF

//all sust charge
IF LCP.Section[1].Sust.ChargeRelay1_close = TRUE AND
	LCP.Section[1].Sust.ChargeRelay2_close = TRUE AND
	LCP.Section[2].Sust.ChargeRelay1_close = TRUE AND
	LCP.Section[2].Sust.ChargeRelay2_close = TRUE AND
	LCP.Section[3].Sust.ChargeRelay1_close = TRUE AND
	LCP.Section[3].Sust.ChargeRelay2_close = TRUE 
	THEN
		Permissives_DB.AllSustChargeRlyClose := TRUE;
		ELSE
			Permissives_DB.AllSustChargeRlyClose := FALSE;
END_IF
//all form charge
IF	LCP.Section[4].Form.ChargeRelay1_close = TRUE AND
	LCP.Section[4].Form.ChargeRelay2_close = TRUE 
	THEN
		Permissives_DB.AllFormChargeRlyClose := TRUE;
		ELSE
			Permissives_DB.AllFormChargeRlyClose := FALSE;
END_IF

//all peak dump
IF LCP.Section[1].Peak.DumpRelay1_close = TRUE AND
	LCP.Section[1].Peak.DumpRelay2_close = TRUE AND
	LCP.Section[2].Peak.DumpRelay1_close = TRUE AND
	LCP.Section[2].Peak.DumpRelay2_close = TRUE AND
	LCP.Section[3].Peak.DumpRelay1_close = TRUE AND
	LCP.Section[3].Peak.DumpRelay2_close = TRUE 
	THEN
		Permissives_DB.AllPeakDumpRlyOpen := FALSE;
		ELSE
			Permissives_DB.AllPeakDumpRlyOpen := TRUE;
END_IF
//all sust dump
IF LCP.Section[1].Sust.DumpRelay1_close = TRUE AND
	LCP.Section[1].Sust.DumpRelay2_close = TRUE AND
	LCP.Section[2].Sust.DumpRelay1_close = TRUE AND
	LCP.Section[2].Sust.DumpRelay2_close = TRUE AND
	LCP.Section[3].Sust.DumpRelay1_close = TRUE AND
	LCP.Section[3].Sust.DumpRelay2_close = TRUE 
	THEN
		Permissives_DB.AllSustDumpRlyOpen := FALSE;
		ELSE
			Permissives_DB.AllSustDumpRlyOpen := TRUE;
END_IF
//all form dump
IF LCP.Section[4].Form.DumpRelay1_close = TRUE AND
	LCP.Section[4].Form.DumpRelay2_close = TRUE 
	THEN
		Permissives_DB.AllFormDumpRlyOpen := FALSE;
		ELSE
			Permissives_DB.AllFormDumpRlyOpen := TRUE;
END_IF
// GLS 1 & 2 can use raw input bit.

//section 1 charge
IF LCP.Section[1].Peak.ChargeRelay1_close = TRUE AND
	LCP.Section[1].Peak.ChargeRelay2_close = TRUE AND
	LCP.Section[1].Sust.ChargeRelay1_close = TRUE AND
	LCP.Section[1].Sust.ChargeRelay2_close = TRUE 
	THEN
		Permissives_DB.AllSection1ChargeRlyClose := TRUE;
		ELSE
			Permissives_DB.AllSection1ChargeRlyClose := FALSE;
END_IF;
//section 2 charge
IF LCP.Section[2].Peak.ChargeRelay1_close = TRUE AND
	LCP.Section[2].Peak.ChargeRelay2_close = TRUE AND
	LCP.Section[2].Sust.ChargeRelay1_close = TRUE AND
	LCP.Section[2].Sust.ChargeRelay2_close = TRUE 
	THEN
		Permissives_DB.AllSection2ChargeRlyClose := TRUE;
		ELSE
			Permissives_DB.AllSection2ChargeRlyClose := FALSE;
END_IF;
//section 3 charge
IF LCP.Section[3].Peak.ChargeRelay1_close = TRUE AND
	LCP.Section[3].Peak.ChargeRelay2_close = TRUE AND
	LCP.Section[3].Sust.ChargeRelay1_close = TRUE AND
	LCP.Section[3].Sust.ChargeRelay2_close = TRUE 
	THEN
		Permissives_DB.AllSection3ChargeRlyClose := TRUE;
		ELSE
			Permissives_DB.AllSection3ChargeRlyClose := FALSE;
END_IF;
//section 4 charge
IF	LCP.Section[4].Form.ChargeRelay1_close = TRUE AND
	LCP.Section[4].Form.ChargeRelay2_close = TRUE AND						
	LCP.Section[4].Form.PreFormChargeRly_close = TRUE AND
	LCP.Section[4].Form.FormTrigChargeRly_close = TRUE AND
	LCP.Section[4].Form.PreFormTrigChargeRly_close = TRUE
	THEN
		Permissives_DB.AllSection4ChargeRlyClose := TRUE;
		ELSE
			Permissives_DB.AllSection4ChargeRlyClose := FALSE;
END_IF
	
//All charge relay close
IF ((LCP.Section[1].Peak.ChargeRelay1_close = TRUE OR Recipe.PeakSupplyEN = FALSE)AND
	(LCP.Section[1].Peak.ChargeRelay2_close = TRUE OR Recipe.PeakSupplyEN = FALSE)AND
	(LCP.Section[1].Sust.ChargeRelay1_close = TRUE OR Recipe.SustSupplyEN = FALSE)AND
	(LCP.Section[1].Sust.ChargeRelay2_close = TRUE OR Recipe.SustSupplyEN = FALSE)AND
	(LCP.Section[2].Peak.ChargeRelay1_close = TRUE OR Recipe.PeakSupplyEN = FALSE)AND
	(LCP.Section[2].Peak.ChargeRelay2_close = TRUE OR Recipe.PeakSupplyEN = FALSE)AND
	(LCP.Section[2].Sust.ChargeRelay1_close = TRUE OR Recipe.SustSupplyEN = FALSE)AND
	(LCP.Section[2].Sust.ChargeRelay2_close = TRUE OR Recipe.SustSupplyEN = FALSE)AND
	(LCP.Section[3].Peak.ChargeRelay1_close = TRUE OR Recipe.PeakSupplyEN = FALSE)AND
	(LCP.Section[3].Peak.ChargeRelay2_close = TRUE OR Recipe.PeakSupplyEN = FALSE)AND
	(LCP.Section[3].Sust.ChargeRelay1_close = TRUE OR Recipe.SustSupplyEN = FALSE)AND
	(LCP.Section[3].Sust.ChargeRelay2_close = TRUE OR Recipe.SustSupplyEN = FALSE)AND
	
	(LCP.Section[4].Form.ChargeRelay1_close = TRUE OR Recipe.FormSupplyEN = FALSE)AND
	(LCP.Section[4].Form.ChargeRelay2_close = TRUE OR Recipe.FormSupplyEN = FALSE)AND						
	(LCP.Section[4].Form.PreFormChargeRly_close = TRUE OR Recipe.PFormSupplyEN = FALSE)AND
	(LCP.Section[4].Form.FormTrigChargeRly_close = TRUE  OR Recipe.FormSupplyEN = FALSE)AND
	(LCP.Section[4].Form.PreFormTrigChargeRly_close = TRUE OR Recipe.PFormSupplyEN = FALSE)) OR HMI_DB.AllChargeRelayCloseBP = TRUE //admin bypass 
	THEN
		Permissives_DB.AllChargeRelaysClosed := TRUE;
	ELSE
		Permissives_DB.AllChargeRelaysClosed := FALSE;
END_IF;

//section 1 dump
IF LCP.Section[1].Peak.DumpRelay1_close = FALSE AND
	LCP.Section[1].Peak.DumpRelay2_close = FALSE AND
	LCP.Section[1].Sust.DumpRelay1_close = FALSE AND
	LCP.Section[1].Sust.DumpRelay2_close = FALSE
	THEN
		Permissives_DB.AllSection1DumpRlyOpen := TRUE;
		ELSE
			Permissives_DB.AllSection1DumpRlyOpen := FALSE;
END_IF
//section 2 dump
IF LCP.Section[2].Peak.DumpRelay1_close = FALSE AND
	LCP.Section[2].Peak.DumpRelay2_close = FALSE AND
	LCP.Section[2].Sust.DumpRelay1_close = FALSE AND
	LCP.Section[2].Sust.DumpRelay2_close = FALSE
	THEN
		Permissives_DB.AllSection2DumpRlyOpen := TRUE;
		ELSE
			Permissives_DB.AllSection2DumpRlyOpen := FALSE;
END_IF
//section 3 dump
IF LCP.Section[3].Peak.DumpRelay1_close = FALSE AND
	LCP.Section[3].Peak.DumpRelay2_close = FALSE AND
	LCP.Section[3].Sust.DumpRelay1_close = FALSE AND
	LCP.Section[3].Sust.DumpRelay2_close = FALSE
	THEN
		Permissives_DB.AllSection3DumpRlyOpen := TRUE;
		ELSE
			Permissives_DB.AllSection3DumpRlyOpen := FALSE;
END_IF
//section 4 dump
IF 	LCP.Section[4].Form.DumpRelay1_close = FALSE AND
	LCP.Section[4].Form.DumpRelay2_close = FALSE AND						
	LCP.Section[4].Form.PreFormDumpRly_close = FALSE AND
	LCP.Section[4].Form.FormTrigDumpRly1_close = FALSE AND
	LCP.Section[4].Form.PreFormTrigDumpRly1_close = FALSE
	THEN
		Permissives_DB.AllSection4DumpRlyOpen := TRUE;
		ELSE
			Permissives_DB.AllSection4DumpRlyOpen := FALSE;
END_IF

